KUKA KRL program: EPS_2_251806_MH01A_A_20260213065128.src

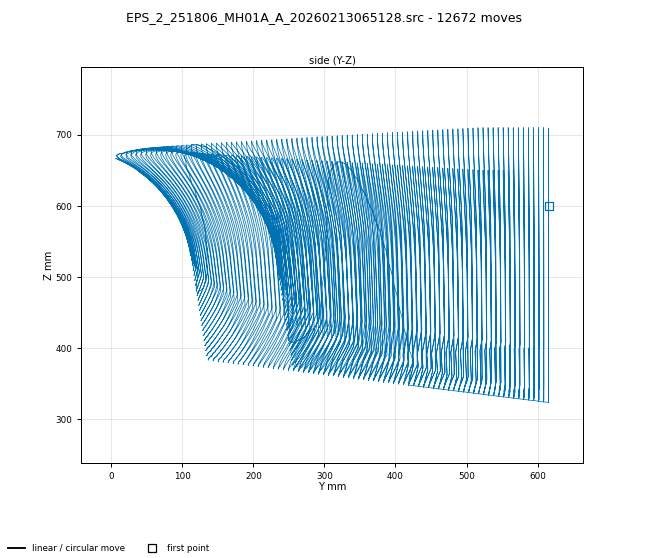
[picture p0: tool path of EPS_2_251806_MH01A_A_20260213065128.src, 12672 of 12674 moves have a stored position in this frame; points joined in program order, loops and branches not executed]
&ACCESS RVP
&REL 4
&COMMENT QRS 19112012
&PARAM EDITMASK = *
DEF PART()
EXT BAS (BAS_COMMAND :IN,REAL :IN )
INT I
BAS (#INITMOV,0 )

;KUKA QRS Post kuka4.cps  Date:22-06-2017 !

File_ID=3009

QRS_PRE_INIT()

;Init var - Until changes are made in qrs_pre_init
Outlet_Square_prg=0
Inlet_1_Square_prg=0
Inlet_2_Square_prg=0
Inlet_3_Square_prg=0
Inlet_4_Square_prg=0
Inlet_5_Square_prg=0

Outlet_1={X 0.000, Y 517.920, Z 561.000, B 0.000, E1 0.000 }
Inlet_1={X 0.000, Y 522.300, Z 501.000, B 0.000, E1 220.000 }
Outlet_1_type=299
Inlet_1_type=299
;QRS#1=Sidecore dimensions
;QRS#2=300-12" PVC SDR 35
;QRS#3=300-12" PVC SDR 35
;QRS#4=
;QRS#5=
;QRS#6=
;QRS#7=
;QRS#8=
;QRS#9=16M PSX
;QRS#10=16M PSX
;QRS#11=
;QRS#12=
;QRS#13=
;QRS#14=
;QRS#15=
;QRS#16=1220x127x991 3,25'
;QRS#17=EPS Height
;QRS#18=710,5
;QRS#19=*
;QRS#20= UPDATED VERSION 22-06-2017
;QRS#21=*
Outlet_Square=0150
Inlet_1_Square=0150
Inlet_2_Square=0
Inlet_3_Square=0
Inlet_4_Square=0
Inlet_5_Square=0
Mill_Square=1
Outlet_Square_Prg=206
Inlet_1_Square_prg=206

QRS_INIT()

$ADVANCE=5

; T1
PTP {E1 173.607,E2 173.607}
PTP {X 0,Y 615.503,A -85,B 0,C 180,E1 173.607,E2 173.607,E3 0,E4 0,E5 0,E6 0}
QRS_SPEED_INIT()
LIN {X 0,Y 615.503,Z 600,A -85,B 0,C 180,E1 173.607,E2 173.607,E3 0,E4 0,E5 0,E6 0} C_VEL
LIN {X 0,Y 615.503,Z 333.492,A -85,B 0,C 180,E1 173.607,E2 173.607} C_VEL
LIN {X 0,Y 615.503,Z 325.319,A -85,B 0,C 180,E1 173.607,E2 173.607} C_VEL
LIN {X 0,Y 615.485,Z 323.319,A -85,B 0,C 180,E1 173.421,E2 173.421} C_VEL
LIN {X 0,Y 615.473,Z 323.319,A -85,B 0,C 180,E1 170.801,E2 170.801} C_VEL
LIN {X 0,Y 615.487,Z 323.307,A -85,B 0,C 180,E1 168.139,E2 168.139} C_VEL
LIN {X 0,Y 615.487,Z 323.319,A -85,B 0,C 180,E1 165.451,E2 165.451} C_VEL
LIN {X 0,Y 615.467,Z 323.317,A -85,B 0,C 180,E1 162.729,E2 162.729} C_VEL
LIN {X 0,Y 615.489,Z 323.308,A -85,B 0,C 180,E1 159.967,E2 159.967} C_VEL
LIN {X 0,Y 615.489,Z 323.324,A -85,B 0,C 180,E1 157.155,E2 157.155} C_VEL
LIN {X 0,Y 615.466,Z 323.312,A -85,B 0,C 180,E1 154.435,E2 154.435} C_VEL
LIN {X 0,Y 615.489,Z 323.319,A -85,B 0,C 180,E1 151.549,E2 151.549} C_VEL
LIN {X 0,Y 615.465,Z 323.32,A -85,B 0,C 180,E1 148.917,E2 148.917} C_VEL
LIN {X 0,Y 615.462,Z 323.313,A -85,B 0,C 180,E1 146.469,E2 146.469} C_VEL
LIN {X 0,Y 615.482,Z 323.309,A -85,B 0,C 180,E1 144.166,E2 144.166} C_VEL
LIN {X 0,Y 615.488,Z 323.311,A -85,B 0,C 180,E1 141.931,E2 141.931} C_VEL
LIN {X 0,Y 615.487,Z 323.328,A -85,B 0,C 180,E1 139.393,E2 139.393} C_VEL
LIN {X 0,Y 615.455,Z 323.317,A -85,B 0,C 180,E1 136.752,E2 136.752} C_VEL
LIN {X 0,Y 615.487,Z 323.311,A -85,B 0,C 180,E1 133.997,E2 133.997} C_VEL
LIN {X 0,Y 615.464,Z 323.321,A -85,B 0,C 180,E1 131.091,E2 131.091} C_VEL
LIN {X 0,Y 615.454,Z 323.319,A -85,B 0,C 180,E1 128.906,E2 128.906} C_VEL
LIN {X 0,Y 615.459,Z 323.314,A -85,B 0,C 180,E1 126.426,E2 126.426} C_VEL
LIN {X 0,Y 615.498,Z 323.324,A -85,B 0,C 180,E1 123.535,E2 123.535} C_VEL
LIN {X 0,Y 615.449,Z 323.319,A -85,B 0,C 180,E1 120.921,E2 120.921} C_VEL
LIN {X 0,Y 615.455,Z 323.315,A -85,B 0,C 180,E1 118.444,E2 118.444} C_VEL
LIN {X 0,Y 615.499,Z 323.325,A -85,B 0,C 180,E1 115.57,E2 115.57} C_VEL
LIN {X 0,Y 615.443,Z 323.319,A -85,B 0,C 180,E1 112.846,E2 112.846} C_VEL
LIN {X 0,Y 615.447,Z 323.316,A -85,B 0,C 180,E1 110.546,E2 110.546} C_VEL
LIN {X 0,Y 615.494,Z 323.315,A -85,B 0,C 180,E1 107.956,E2 107.956} C_VEL
LIN {X 0,Y 615.455,Z 323.322,A -85,B 0,C 180,E1 105.227,E2 105.227} C_VEL
LIN {X 0,Y 615.451,Z 323.322,A -85,B 0,C 180,E1 103.202,E2 103.202} C_VEL
LIN {X 0,Y 615.434,Z 323.32,A -85,B 0,C 180,E1 100.86,E2 100.86} C_VEL
LIN {X 0,Y 615.444,Z 323.317,A -85,B 0,C 180,E1 98.537,E2 98.537} C_VEL
LIN {X 0,Y 615.497,Z 323.318,A -85,B 0,C 180,E1 95.898,E2 95.898} C_VEL
LIN {X 0,Y 615.448,Z 323.323,A -85,B 0,C 180,E1 93.273,E2 93.273} C_VEL
LIN {X 0,Y 615.449,Z 323.323,A -85,B 0,C 180,E1 91.308,E2 91.308} C_VEL
LIN {X 0,Y 615.451,Z 323.323,A -85,B 0,C 180,E1 89.345,E2 89.345} C_VEL
LIN {X 0,Y 615.452,Z 323.323,A -85,B 0,C 180,E1 87.382,E2 87.382} C_VEL
LIN {X 0,Y 615.454,Z 323.323,A -85,B 0,C 180,E1 85.415,E2 85.415} C_VEL
LIN {X 0,Y 615.455,Z 323.324,A -85,B 0,C 180,E1 83.443,E2 83.443} C_VEL
LIN {X 0,Y 615.455,Z 323.324,A -85,B 0,C 180,E1 81.463,E2 81.463} C_VEL
LIN {X 0,Y 615.429,Z 323.323,A -85,B 0,C 180,E1 79.143,E2 79.143} C_VEL
LIN {X 0,Y 615.424,Z 323.322,A -85,B 0,C 180,E1 76.797,E2 76.797} C_VEL
LIN {X 0,Y 615.479,Z 323.321,A -85,B 0,C 180,E1 74.094,E2 74.094} C_VEL
LIN {X 0,Y 615.435,Z 323.324,A -85,B 0,C 180,E1 71.352,E2 71.352} C_VEL
LIN {X 0,Y 615.433,Z 323.469,A -85,B 0,C 180,E1 70.552,E2 70.552} C_VEL
LIN {X 0,Y 615.467,Z 340.354,A -85,B 0,C 180,E1 68.193,E2 68.193} C_VEL
LIN {X 0,Y 615.47,Z 505.061,A -85,B 0,C 180,E1 66.189,E2 66.189} C_VEL
LIN {X 0,Y 615.489,Z 520.711,A -85,B 0,C 180,E1 65.86,E2 65.86} C_VEL
LIN {X 0,Y 615.479,Z 535.48,A -85,B 0,C 180,E1 65.413,E2 65.413} C_VEL
LIN {X 0,Y 615.487,Z 549.225,A -85,B 0,C 180,E1 64.865,E2 64.865} C_VEL
LIN {X 0,Y 615.482,Z 562.727,A -85,B 0,C 180,E1 64.193,E2 64.193} C_VEL
LIN {X 0,Y 615.496,Z 575.661,A -85,B 0,C 180,E1 63.406,E2 63.406} C_VEL
LIN {X 0,Y 615.494,Z 587.419,A -85,B 0,C 180,E1 62.547,E2 62.547} C_VEL
LIN {X 0,Y 615.496,Z 598.891,A -85,B 0,C 180,E1 61.549,E2 61.549} C_VEL
LIN {X 0,Y 615.495,Z 609.92,A -85,B 0,C 180,E1 60.399,E2 60.399} C_VEL
LIN {X 0,Y 615.497,Z 618.936,A -85,B 0,C 180,E1 59.271,E2 59.271} C_VEL
LIN {X 0,Y 615.493,Z 627.407,A -85,B 0,C 180,E1 57.992,E2 57.992} C_VEL
LIN {X 0,Y 615.493,Z 634.042,A -85,B 0,C 180,E1 56.764,E2 56.764} C_VEL
LIN {X 0,Y 615.496,Z 639.007,A -85,B 0,C 180,E1 55.64,E2 55.64} C_VEL
LIN {X 0,Y 615.496,Z 643.984,A -85,B 0,C 180,E1 54.166,E2 54.166} C_VEL
LIN {X 0,Y 615.491,Z 647.294,A -85,B 0,C 180,E1 52.758,E2 52.758} C_VEL
LIN {X 0,Y 615.495,Z 648.577,A -85,B 0,C 180,E1 51.932,E2 51.932} C_VEL
LIN {X 0,Y 615.49,Z 649.536,A -85,B 0,C 180,E1 50.938,E2 50.938} C_VEL
LIN {X 0,Y 615.498,Z 649.883,A -85,B 0,C 180,E1 49.91,E2 49.91} C_VEL
LIN {X 0,Y 615.491,Z 649.219,A -85,B 0,C 180,E1 48.526,E2 48.526} C_VEL
LIN {X 0,Y 615.49,Z 646.908,A -85,B 0,C 180,E1 46.953,E2 46.953} C_VEL
LIN {X 0,Y 615.493,Z 643.15,A -85,B 0,C 180,E1 45.461,E2 45.461} C_VEL
LIN {X 0,Y 615.496,Z 638.541,A -85,B 0,C 180,E1 44.149,E2 44.149} C_VEL
LIN {X 0,Y 615.49,Z 631.812,A -85,B 0,C 180,E1 42.7,E2 42.7} C_VEL
LIN {X 0,Y 615.494,Z 624.699,A -85,B 0,C 180,E1 41.474,E2 41.474} C_VEL
LIN {X 0,Y 615.496,Z 615.8,A -85,B 0,C 180,E1 40.219,E2 40.219} C_VEL
LIN {X 0,Y 615.495,Z 605.897,A -85,B 0,C 180,E1 39.063,E2 39.063} C_VEL
LIN {X 0,Y 615.496,Z 595.149,A -85,B 0,C 180,E1 38.013,E2 38.013} C_VEL
LIN {X 0,Y 615.495,Z 582.892,A -85,B 0,C 180,E1 37.013,E2 37.013} C_VEL
LIN {X 0,Y 615.497,Z 569.807,A -85,B 0,C 180,E1 36.129,E2 36.129} C_VEL
LIN {X 0,Y 615.476,Z 556.032,A -85,B 0,C 180,E1 35.366,E2 35.366} C_VEL
LIN {X 0,Y 615.492,Z 542.424,A -85,B 0,C 180,E1 34.758,E2 34.758} C_VEL
LIN {X 0,Y 615.486,Z 527.304,A -85,B 0,C 180,E1 34.234,E2 34.234} C_VEL
LIN {X 0,Y 615.48,Z 512.906,A -85,B 0,C 180,E1 33.868,E2 33.868} C_VEL
LIN {X 0,Y 615.461,Z 496.852,A -85,B 0,C 180,E1 33.605,E2 33.605} C_VEL
LIN {X 0,Y 615.465,Z 340.427,A -85,B 0,C 180,E1 31.727,E2 31.727} C_VEL
LIN {X 0,Y 615.421,Z 323.324,A -85,B 0,C 180,E1 29.328,E2 29.328} C_VEL
LIN {X 0,Y 615.415,Z 323.324,A -85,B 0,C 180,E1 27.031,E2 27.031} C_VEL
LIN {X 0,Y 615.475,Z 323.325,A -85,B 0,C 180,E1 24.273,E2 24.273} C_VEL
LIN {X 0,Y 615.433,Z 323.321,A -85,B 0,C 180,E1 21.434,E2 21.434} C_VEL
LIN {X 0,Y 615.43,Z 323.321,A -85,B 0,C 180,E1 19.34,E2 19.34} C_VEL
LIN {X 0,Y 615.429,Z 323.321,A -85,B 0,C 180,E1 17.272,E2 17.272} C_VEL
LIN {X 0,Y 615.43,Z 323.32,A -85,B 0,C 180,E1 15.228,E2 15.228} C_VEL
LIN {X 0,Y 615.432,Z 323.32,A -85,B 0,C 180,E1 13.203,E2 13.203} C_VEL
LIN {X 0,Y 615.47,Z 323.324,A -85,B 0,C 180,E1 10.527,E2 10.527} C_VEL
LIN {X 0,Y 615.48,Z 323.315,A -85,B 0,C 180,E1 7.876,E2 7.876} C_VEL
LIN {X 0,Y 615.439,Z 323.319,A -85,B 0,C 180,E1 5.242,E2 5.242} C_VEL
LIN {X 0,Y 615.475,Z 323.323,A -85,B 0,C 180,E1 2.618,E2 2.618} C_VEL
LIN {X 0,Y 615.486,Z 323.314,A -85,B 0,C 180,E1 0,E2 0} C_VEL
LIN {X 0,Y 615.45,Z 323.316,A -85,B 0,C 180,E1 -2.618,E2 -2.618} C_VEL
LIN {X 0,Y 615.474,Z 323.323,A -85,B 0,C 180,E1 -5.241,E2 -5.241} C_VEL
LIN {X 0,Y 615.493,Z 323.313,A -85,B 0,C 180,E1 -7.875,E2 -7.875} C_VEL
LIN {X 0,Y 615.458,Z 323.314,A -85,B 0,C 180,E1 -10.527,E2 -10.527} C_VEL
LIN {X 0,Y 615.483,Z 323.323,A -85,B 0,C 180,E1 -13.201,E2 -13.201} C_VEL
LIN {X 0,Y 615.491,Z 323.31,A -85,B 0,C 180,E1 -15.905,E2 -15.905} C_VEL
LIN {X 0,Y 615.462,Z 323.316,A -85,B 0,C 180,E1 -18.647,E2 -18.647} C_VEL
LIN {X 0,Y 615.489,Z 323.321,A -85,B 0,C 180,E1 -21.432,E2 -21.432} C_VEL
LIN {X 0,Y 615.477,Z 323.31,A -85,B 0,C 180,E1 -24.272,E2 -24.272} C_VEL
LIN {X 0,Y 615.487,Z 323.328,A -85,B 0,C 180,E1 -27.177,E2 -27.177} C_VEL
LIN {X 0,Y 615.486,Z 323.308,A -85,B 0,C 180,E1 -30.16,E2 -30.16} C_VEL
LIN {X 0,Y 615.474,Z 323.313,A -85,B 0,C 180,E1 -32.458,E2 -32.458} C_VEL
LIN {X 0,Y 615.477,Z 323.322,A -85,B 0,C 180,E1 -34.816,E2 -34.816} C_VEL
LIN {X 0,Y 615.485,Z 323.321,A -85,B 0,C 180,E1 -37.242,E2 -37.242} C_VEL
LIN {X 0,Y 615.493,Z 323.306,A -85,B 0,C 180,E1 -40.089,E2 -40.089} C_VEL
LIN {X 0,Y 615.49,Z 323.323,A -85,B 0,C 180,E1 -43.047,E2 -43.047} C_VEL
LIN {X 0,Y 615.487,Z 323.308,A -85,B 0,C 180,E1 -46.002,E2 -46.002} C_VEL
LIN {X 0,Y 615.485,Z 323.327,A -85,B 0,C 180,E1 -48.906,E2 -48.906} C_VEL
LIN {X 0,Y 615.478,Z 323.321,A -85,B 0,C 180,E1 -51.095,E2 -51.095} C_VEL
LIN {X 0,Y 615.469,Z 323.312,A -85,B 0,C 180,E1 -53.574,E2 -53.574} C_VEL
LIN {X 0,Y 615.488,Z 323.318,A -85,B 0,C 180,E1 -56.466,E2 -56.466} C_VEL
LIN {X 0,Y 615.469,Z 323.32,A -85,B 0,C 180,E1 -59.079,E2 -59.079} C_VEL
LIN {X 0,Y 615.464,Z 323.313,A -85,B 0,C 180,E1 -61.554,E2 -61.554} C_VEL
LIN {X 0,Y 615.478,Z 323.359,A -85,B 0,C 180,E1 -63.783,E2 -63.783} C_VEL
LIN {X 0,Y 615.479,Z 349.6,A -85,B 0,C 180,E1 -66.621,E2 -66.621} C_VEL
LIN {X 0,Y 615.488,Z 376.247,A -85,B 0,C 180,E1 -69.443,E2 -69.443} C_VEL
LIN {X 0,Y 615.496,Z 398.316,A -85,B 0,C 180,E1 -71.741,E2 -71.741} C_VEL
LIN {X 0,Y 615.481,Z 565.27,A -85,B 0,C 180,E1 -73.77,E2 -73.77} C_VEL
LIN {X 0,Y 615.49,Z 580.703,A -85,B 0,C 180,E1 -74.095,E2 -74.095} C_VEL
LIN {X 0,Y 615.48,Z 596.043,A -85,B 0,C 180,E1 -74.562,E2 -74.562} C_VEL
LIN {X 0,Y 615.484,Z 609.747,A -85,B 0,C 180,E1 -75.112,E2 -75.112} C_VEL
LIN {X 0,Y 615.493,Z 624.044,A -85,B 0,C 180,E1 -75.833,E2 -75.833} C_VEL
LIN {X 0,Y 615.497,Z 636.895,A -85,B 0,C 180,E1 -76.631,E2 -76.631} C_VEL
LIN {X 0,Y 615.495,Z 649.252,A -85,B 0,C 180,E1 -77.554,E2 -77.554} C_VEL
LIN {X 0,Y 615.495,Z 659.604,A -85,B 0,C 180,E1 -78.473,E2 -78.473} C_VEL
LIN {X 0,Y 615.494,Z 669.182,A -85,B 0,C 180,E1 -79.473,E2 -79.473} C_VEL
LIN {X 0,Y 615.493,Z 678.575,A -85,B 0,C 180,E1 -80.635,E2 -80.635} C_VEL
LIN {X 0,Y 615.497,Z 686.379,A -85,B 0,C 180,E1 -81.794,E2 -81.794} C_VEL
LIN {X 0,Y 615.494,Z 693.609,A -85,B 0,C 180,E1 -83.102,E2 -83.102} C_VEL
LIN {X 0,Y 615.499,Z 699.435,A -85,B 0,C 180,E1 -84.43,E2 -84.43} C_VEL
LIN {X 0,Y 615.491,Z 702.859,A -85,B 0,C 180,E1 -85.415,E2 -85.415} C_VEL
LIN {X 0,Y 615.493,Z 706.317,A -85,B 0,C 180,E1 -86.727,E2 -86.727} C_VEL
LIN {X 0,Y 615.499,Z 708.592,A -85,B 0,C 180,E1 -88.037,E2 -88.037} C_VEL
LIN {X 0,Y 615.491,Z 709.741,A -85,B 0,C 180,E1 -89.345,E2 -89.345} C_VEL
LIN {X 0,Y 615.491,Z 709.741,A -85,B 0,C 180,E1 -90.654,E2 -90.654} C_VEL
LIN {X 0,Y 615.499,Z 708.593,A -85,B 0,C 180,E1 -91.963,E2 -91.963} C_VEL
LIN {X 0,Y 615.493,Z 706.319,A -85,B 0,C 180,E1 -93.273,E2 -93.273} C_VEL
LIN {X 0,Y 615.491,Z 702.861,A -85,B 0,C 180,E1 -94.584,E2 -94.584} C_VEL
LIN {X 0,Y 615.497,Z 698.144,A -85,B 0,C 180,E1 -95.898,E2 -95.898} C_VEL
LIN {X 0,Y 615.492,Z 692.031,A -85,B 0,C 180,E1 -97.215,E2 -97.215} C_VEL
LIN {X 0,Y 615.49,Z 684.335,A -85,B 0,C 180,E1 -98.536,E2 -98.536} C_VEL
LIN {X 0,Y 615.495,Z 676.116,A -85,B 0,C 180,E1 -99.696,E2 -99.696} C_VEL
LIN {X 0,Y 615.496,Z 665.898,A -85,B 0,C 180,E1 -100.892,E2 -100.892} C_VEL
LIN {X 0,Y 615.496,Z 656.07,A -85,B 0,C 180,E1 -101.86,E2 -101.86} C_VEL
LIN {X 0,Y 615.497,Z 643.951,A -85,B 0,C 180,E1 -102.865,E2 -102.865} C_VEL
LIN {X 0,Y 615.498,Z 631.802,A -85,B 0,C 180,E1 -103.705,E2 -103.705} C_VEL
LIN {X 0,Y 615.477,Z 618.384,A -85,B 0,C 180,E1 -104.472,E2 -104.472} C_VEL
LIN {X 0,Y 615.495,Z 603.855,A -85,B 0,C 180,E1 -105.141,E2 -105.141} C_VEL
LIN {X 0,Y 615.48,Z 589.625,A -85,B 0,C 180,E1 -105.65,E2 -105.65} C_VEL
LIN {X 0,Y 615.5,Z 575.177,A -85,B 0,C 180,E1 -106.035,E2 -106.035} C_VEL
LIN {X 0,Y 615.478,Z 560.741,A -85,B 0,C 180,E1 -106.296,E2 -106.296} C_VEL
LIN {X 0,Y 615.495,Z 398.319,A -85,B 0,C 180,E1 -108.259,E2 -108.259} C_VEL
LIN {X 0,Y 615.484,Z 372.931,A -85,B 0,C 180,E1 -110.905,E2 -110.905} C_VEL
LIN {X 0,Y 615.477,Z 346.881,A -85,B 0,C 180,E1 -113.67,E2 -113.67} C_VEL
LIN {X 0,Y 615.477,Z 323.365,A -85,B 0,C 180,E1 -116.216,E2 -116.216} C_VEL
LIN {X 0,Y 615.458,Z 323.316,A -85,B 0,C 180,E1 -118.659,E2 -118.659} C_VEL
LIN {X 0,Y 615.476,Z 323.322,A -85,B 0,C 180,E1 -121.084,E2 -121.084} C_VEL
LIN {X 0,Y 615.492,Z 323.308,A -85,B 0,C 180,E1 -124.021,E2 -124.021} C_VEL
LIN {X 0,Y 615.466,Z 323.312,A -85,B 0,C 180,E1 -126.426,E2 -126.426} C_VEL
LIN {X 0,Y 615.48,Z 323.322,A -85,B 0,C 180,E1 -129.061,E2 -129.061} C_VEL
LIN {X 0,Y 615.489,Z 323.319,A -85,B 0,C 180,E1 -131.473,E2 -131.473} C_VEL
LIN {X 0,Y 615.485,Z 323.308,A -85,B 0,C 180,E1 -134.149,E2 -134.149} C_VEL
LIN {X 0,Y 615.477,Z 323.321,A -85,B 0,C 180,E1 -136.953,E2 -136.953} C_VEL
LIN {X 0,Y 615.494,Z 323.307,A -85,B 0,C 180,E1 -139.91,E2 -139.91} C_VEL
LIN {X 0,Y 615.471,Z 323.318,A -85,B 0,C 180,E1 -142.757,E2 -142.757} C_VEL
LIN {X 0,Y 615.491,Z 323.322,A -85,B 0,C 180,E1 -145.298,E2 -145.298} C_VEL
LIN {X 0,Y 615.481,Z 323.313,A -85,B 0,C 180,E1 -147.669,E2 -147.669} C_VEL
LIN {X 0,Y 615.483,Z 323.308,A -85,B 0,C 180,E1 -150.205,E2 -150.205} C_VEL
LIN {X 0,Y 615.488,Z 323.322,A -85,B 0,C 180,E1 -152.954,E2 -152.954} C_VEL
LIN {X 0,Y 615.484,Z 323.31,A -85,B 0,C 180,E1 -155.728,E2 -155.728} C_VEL
LIN {X 0,Y 615.474,Z 323.316,A -85,B 0,C 180,E1 -158.568,E2 -158.568} C_VEL
LIN {X 0,Y 615.48,Z 323.317,A -85,B 0,C 180,E1 -161.396,E2 -161.396} C_VEL
LIN {X 0,Y 615.487,Z 323.307,A -85,B 0,C 180,E1 -164.095,E2 -164.095} C_VEL
LIN {X 0,Y 615.484,Z 323.321,A -85,B 0,C 180,E1 -166.799,E2 -166.799} C_VEL
LIN {X 0,Y 615.476,Z 323.315,A -85,B 0,C 180,E1 -169.473,E2 -169.473} C_VEL
LIN {X 0,Y 615.488,Z 323.307,A -85,B 0,C 180,E1 -172.125,E2 -172.125} C_VEL
LIN {X 0,Y 615.485,Z 323.322,A -85,B 0,C 180,E1 -174.759,E2 -174.759} C_VEL
LIN {X 0,Y 615.474,Z 323.316,A -85,B 0,C 180,E1 -177.382,E2 -177.382} C_VEL
LIN {X 0,Y 615.486,Z 323.308,A -85,B 0,C 180,E1 -180,E2 -180} C_VEL
LIN {X 0,Y 615.483,Z 323.319,A -85,B 0,C 180,E1 -182.618,E2 -182.618} C_VEL
LIN {X 0,Y 615.474,Z 323.318,A -85,B 0,C 180,E1 -185.242,E2 -185.242} C_VEL
LIN {X 0,Y 615.485,Z 323.319,A -85,B 0,C 180,E1 -186.579,E2 -186.579} C_VEL
LIN {X 0,Y 614.801,Z 323.467,A -85,B 0,C 180,E1 -187.125,E2 -187.125} C_VEL
LIN {X 0,Y 611.96,Z 323.875,A -85,B 0,C 180,E1 -188.011,E2 -188.011} C_VEL
LIN {X 0,Y 609.569,Z 324.187,A -85,B 0,C 180,E1 -188.724,E2 -188.724} C_VEL
LIN {X 0,Y 608.539,Z 324.305,A -85,B 0,C 180,E1 -189.274,E2 -189.274} C_VEL
LIN {X 0,Y 608.452,Z 324.314,A -85,B 0,C 180,E1 -189.46,E2 -189.46} C_VEL
LIN {X 0,Y 608.462,Z 324.311,A -85,B 0,C 180,E1 -192,E2 -192} C_VEL
LIN {X 0,Y 608.471,Z 324.319,A -85,B 0,C 180,E1 -194.721,E2 -194.721} C_VEL
LIN {X 0,Y 608.442,Z 324.314,A -85,B 0,C 180,E1 -197.477,E2 -197.477} C_VEL
LIN {X 0,Y 608.463,Z 324.314,A -85,B 0,C 180,E1 -200.274,E2 -200.274} C_VEL
LIN {X 0,Y 608.445,Z 324.317,A -85,B 0,C 180,E1 -203.125,E2 -203.125} C_VEL
LIN {X 0,Y 608.457,Z 324.312,A -85,B 0,C 180,E1 -205.719,E2 -205.719} C_VEL
LIN {X 0,Y 608.475,Z 324.319,A -85,B 0,C 180,E1 -208.621,E2 -208.621} C_VEL
LIN {X 0,Y 608.439,Z 324.315,A -85,B 0,C 180,E1 -211.319,E2 -211.319} C_VEL
LIN {X 0,Y 608.445,Z 324.313,A -85,B 0,C 180,E1 -213.732,E2 -213.732} C_VEL
LIN {X 0,Y 608.477,Z 324.311,A -85,B 0,C 180,E1 -216.091,E2 -216.091} C_VEL
LIN {X 0,Y 608.462,Z 324.321,A -85,B 0,C 180,E1 -218.589,E2 -218.589} C_VEL
LIN {X 0,Y 608.437,Z 324.315,A -85,B 0,C 180,E1 -221.34,E2 -221.34} C_VEL
LIN {X 0,Y 608.46,Z 324.316,A -85,B 0,C 180,E1 -224.265,E2 -224.265} C_VEL
LIN {X 0,Y 608.43,Z 324.318,A -85,B 0,C 180,E1 -227.039,E2 -227.039} C_VEL
LIN {X 0,Y 608.454,Z 324.312,A -85,B 0,C 180,E1 -229.697,E2 -229.697} C_VEL
LIN {X 0,Y 608.464,Z 324.317,A -85,B 0,C 180,E1 -232.254,E2 -232.254} C_VEL
LIN {X 0,Y 608.42,Z 324.318,A -85,B 0,C 180,E1 -235.099,E2 -235.099} C_VEL
LIN {X 0,Y 608.436,Z 324.314,A -85,B 0,C 180,E1 -237.482,E2 -237.482} C_VEL
LIN {X 0,Y 608.479,Z 324.315,A -85,B 0,C 180,E1 -240.221,E2 -240.221} C_VEL
LIN {X 0,Y 608.416,Z 324.317,A -85,B 0,C 180,E1 -243.225,E2 -243.225} C_VEL
LIN {X 0,Y 608.431,Z 324.315,A -85,B 0,C 180,E1 -245.428,E2 -245.428} C_VEL
LIN {X 0,Y 608.464,Z 324.32,A -85,B 0,C 180,E1 -248.309,E2 -248.309} C_VEL
LIN {X 0,Y 608.436,Z 324.315,A -85,B 0,C 180,E1 -251.13,E2 -251.13} C_VEL
LIN {X 0,Y 608.454,Z 324.315,A -85,B 0,C 180,E1 -253.906,E2 -253.906} C_VEL
LIN {X 0,Y 608.44,Z 324.319,A -85,B 0,C 180,E1 -256.643,E2 -256.643} C_VEL
LIN {X 0,Y 608.406,Z 324.319,A -85,B 0,C 180,E1 -259.078,E2 -259.078} C_VEL
LIN {X 0,Y 608.419,Z 324.316,A -85,B 0,C 180,E1 -261.364,E2 -261.364} C_VEL
LIN {X 0,Y 608.464,Z 324.317,A -85,B 0,C 180,E1 -264.033,E2 -264.033} C_VEL
LIN {X 0,Y 608.42,Z 324.32,A -85,B 0,C 180,E1 -266.689,E2 -266.689} C_VEL
LIN {X 0,Y 608.438,Z 324.318,A -85,B 0,C 180,E1 -268.677,E2 -268.677} C_VEL
LIN {X 0,Y 608.449,Z 324.317,A -85,B 0,C 180,E1 -270.662,E2 -270.662} C_VEL
LIN {X 0,Y 608.403,Z 324.318,A -85,B 0,C 180,E1 -273.311,E2 -273.311} C_VEL
LIN {X 0,Y 608.455,Z 324.318,A -85,B 0,C 180,E1 -275.967,E2 -275.967} C_VEL
LIN {X 0,Y 608.425,Z 324.319,A -85,B 0,C 180,E1 -278.637,E2 -278.637} C_VEL
LIN {X 0,Y 608.413,Z 324.317,A -85,B 0,C 180,E1 -281.325,E2 -281.325} C_VEL
LIN {X 0,Y 608.474,Z 324.318,A -85,B 0,C 180,E1 -284.038,E2 -284.038} C_VEL
LIN {X 0,Y 608.412,Z 324.319,A -85,B 0,C 180,E1 -286.785,E2 -286.785} C_VEL
LIN {X 0,Y 608.431,Z 324.391,A -85,B 0,C 180,E1 -289.33,E2 -289.33} C_VEL
LIN {X 0,Y 608.497,Z 340.471,A -85,B 0,C 180,E1 -291.602,E2 -291.602} C_VEL
LIN {X 0,Y 608.726,Z 347.856,A -85,B 0,C 180,E1 -291.704,E2 -291.704} C_VEL
LIN {X 0,Y 608.67,Z 504.169,A -85,B 0,C 180,E1 -293.611,E2 -293.611} C_VEL
LIN {X 0,Y 608.67,Z 519.292,A -85,B 0,C 180,E1 -293.922,E2 -293.922} C_VEL
LIN {X 0,Y 608.621,Z 534.552,A -85,B 0,C 180,E1 -294.377,E2 -294.377} C_VEL
LIN {X 0,Y 608.595,Z 548.477,A -85,B 0,C 180,E1 -294.93,E2 -294.93} C_VEL
LIN {X 0,Y 608.549,Z 562.697,A -85,B 0,C 180,E1 -295.639,E2 -295.639} C_VEL
LIN {X 0,Y 608.539,Z 575.141,A -85,B 0,C 180,E1 -296.4,E2 -296.4} C_VEL
LIN {X 0,Y 608.529,Z 587.705,A -85,B 0,C 180,E1 -297.323,E2 -297.323} C_VEL
LIN {X 0,Y 608.485,Z 598.502,A -85,B 0,C 180,E1 -298.265,E2 -298.265} C_VEL
LIN {X 0,Y 608.484,Z 609.414,A -85,B 0,C 180,E1 -299.398,E2 -299.398} C_VEL
LIN {X 0,Y 608.453,Z 618.668,A -85,B 0,C 180,E1 -300.546,E2 -300.546} C_VEL
LIN {X 0,Y 608.462,Z 626.497,A -85,B 0,C 180,E1 -301.705,E2 -301.705} C_VEL
LIN {X 0,Y 608.443,Z 633.127,A -85,B 0,C 180,E1 -302.881,E2 -302.881} C_VEL
LIN {X 0,Y 608.44,Z 638.579,A -85,B 0,C 180,E1 -304.071,E2 -304.071} C_VEL
LIN {X 0,Y 608.424,Z 642.975,A -85,B 0,C 180,E1 -305.279,E2 -305.279} C_VEL
LIN {X 0,Y 608.424,Z 645.349,A -85,B 0,C 180,E1 -306.094,E2 -306.094} C_VEL
LIN {X 0,Y 608.432,Z 647.777,A -85,B 0,C 180,E1 -307.153,E2 -307.153} C_VEL
LIN {X 0,Y 608.413,Z 649.814,A -85,B 0,C 180,E1 -308.592,E2 -308.592} C_VEL
LIN {X 0,Y 608.412,Z 650.365,A -85,B 0,C 180,E1 -309.444,E2 -309.444} C_VEL
LIN {X 0,Y 608.437,Z 650.44,A -85,B 0,C 180,E1 -310.327,E2 -310.327} C_VEL
LIN {X 0,Y 608.415,Z 649.935,A -85,B 0,C 180,E1 -311.337,E2 -311.337} C_VEL
LIN {X 0,Y 608.434,Z 648.787,A -85,B 0,C 180,E1 -312.331,E2 -312.331} C_VEL
LIN {X 0,Y 608.433,Z 646.997,A -85,B 0,C 180,E1 -313.305,E2 -313.305} C_VEL
LIN {X 0,Y 608.423,Z 643.011,A -85,B 0,C 180,E1 -314.799,E2 -314.799} C_VEL
LIN {X 0,Y 608.431,Z 638.119,A -85,B 0,C 180,E1 -316.127,E2 -316.127} C_VEL
LIN {X 0,Y 608.438,Z 632.233,A -85,B 0,C 180,E1 -317.38,E2 -317.38} C_VEL
LIN {X 0,Y 608.443,Z 624.795,A -85,B 0,C 180,E1 -318.66,E2 -318.66} C_VEL
LIN {X 0,Y 608.474,Z 615.89,A -85,B 0,C 180,E1 -319.915,E2 -319.915} C_VEL
LIN {X 0,Y 608.494,Z 606.133,A -85,B 0,C 180,E1 -321.058,E2 -321.058} C_VEL
LIN {X 0,Y 608.497,Z 595.21,A -85,B 0,C 180,E1 -322.132,E2 -322.132} C_VEL
LIN {X 0,Y 608.519,Z 583.62,A -85,B 0,C 180,E1 -323.089,E2 -323.089} C_VEL
LIN {X 0,Y 608.548,Z 571.328,A -85,B 0,C 180,E1 -323.942,E2 -323.942} C_VEL
LIN {X 0,Y 608.576,Z 557.514,A -85,B 0,C 180,E1 -324.731,E2 -324.731} C_VEL
LIN {X 0,Y 608.622,Z 543.682,A -85,B 0,C 180,E1 -325.368,E2 -325.368} C_VEL
LIN {X 0,Y 608.637,Z 529.142,A -85,B 0,C 180,E1 -325.892,E2 -325.892} C_VEL
LIN {X 0,Y 608.654,Z 513.527,A -85,B 0,C 180,E1 -326.304,E2 -326.304} C_VEL
LIN {X 0,Y 608.658,Z 497.334,A -85,B 0,C 180,E1 -326.577,E2 -326.577} C_VEL
LIN {X 0,Y 608.598,Z 341.195,A -85,B 0,C 180,E1 -328.471,E2 -328.471} C_VEL
LIN {X 0,Y 608.47,Z 340.371,A -85,B 0,C 180,E1 -328.503,E2 -328.503} C_VEL
LIN {X 0,Y 608.414,Z 324.367,A -85,B 0,C 180,E1 -330.764,E2 -330.764} C_VEL
LIN {X 0,Y 608.391,Z 324.321,A -85,B 0,C 180,E1 -333.223,E2 -333.223} C_VEL
LIN {X 0,Y 608.456,Z 324.323,A -85,B 0,C 180,E1 -335.853,E2 -335.853} C_VEL
LIN {X 0,Y 608.441,Z 324.317,A -85,B 0,C 180,E1 -338.307,E2 -338.307} C_VEL
LIN {X 0,Y 608.428,Z 324.316,A -85,B 0,C 180,E1 -341.129,E2 -341.129} C_VEL
LIN {X 0,Y 608.454,Z 324.321,A -85,B 0,C 180,E1 -343.906,E2 -343.906} C_VEL
LIN {X 0,Y 608.424,Z 324.316,A -85,B 0,C 180,E1 -346.642,E2 -346.642} C_VEL
LIN {X 0,Y 608.439,Z 324.319,A -85,B 0,C 180,E1 -349.349,E2 -349.349} C_VEL
LIN {X 0,Y 608.472,Z 324.314,A -85,B 0,C 180,E1 -352.033,E2 -352.033} C_VEL
LIN {X 0,Y 608.425,Z 324.316,A -85,B 0,C 180,E1 -354.698,E2 -354.698} C_VEL
LIN {X 0,Y 608.465,Z 324.317,A -85,B 0,C 180,E1 -357.352,E2 -357.352} C_VEL
LIN {X 0,Y 608.477,Z 324.313,A -85,B 0,C 180,E1 -360,E2 -360} C_VEL
LIN {X 0,Y 608.445,Z 324.313,A -85,B 0,C 180,E1 -362.648,E2 -362.648} C_VEL
LIN {X 0,Y 608.456,Z 324.32,A -85,B 0,C 180,E1 -365.302,E2 -365.302} C_VEL
LIN {X 0,Y 608.48,Z 324.311,A -85,B 0,C 180,E1 -367.967,E2 -367.967} C_VEL
LIN {X 0,Y 608.438,Z 324.315,A -85,B 0,C 180,E1 -370.65,E2 -370.65} C_VEL
LIN {X 0,Y 608.463,Z 324.322,A -85,B 0,C 180,E1 -373.356,E2 -373.356} C_VEL
LIN {X 0,Y 608.456,Z 324.312,A -85,B 0,C 180,E1 -376.094,E2 -376.094} C_VEL
LIN {X 0,Y 608.448,Z 324.317,A -85,B 0,C 180,E1 -378.87,E2 -378.87} C_VEL
LIN {X 0,Y 608.471,Z 324.313,A -85,B 0,C 180,E1 -381.691,E2 -381.691} C_VEL
LIN {X 0,Y 608.448,Z 324.314,A -85,B 0,C 180,E1 -384.571,E2 -384.571} C_VEL
LIN {X 0,Y 608.481,Z 324.319,A -85,B 0,C 180,E1 -387.207,E2 -387.207} C_VEL
LIN {X 0,Y 608.468,Z 324.311,A -85,B 0,C 180,E1 -389.971,E2 -389.971} C_VEL
LIN {X 0,Y 608.452,Z 324.319,A -85,B 0,C 180,E1 -392.88,E2 -392.88} C_VEL
LIN {X 0,Y 608.437,Z 324.321,A -85,B 0,C 180,E1 -395.278,E2 -395.278} C_VEL
LIN {X 0,Y 608.469,Z 324.311,A -85,B 0,C 180,E1 -397.746,E2 -397.746} C_VEL
LIN {X 0,Y 608.451,Z 324.314,A -85,B 0,C 180,E1 -400.329,E2 -400.329} C_VEL
LIN {X 0,Y 608.456,Z 324.323,A -85,B 0,C 180,E1 -402.959,E2 -402.959} C_VEL
LIN {X 0,Y 608.457,Z 324.312,A -85,B 0,C 180,E1 -405.736,E2 -405.736} C_VEL
LIN {X 0,Y 608.46,Z 324.319,A -85,B 0,C 180,E1 -408.658,E2 -408.658} C_VEL
LIN {X 0,Y 608.436,Z 324.316,A -85,B 0,C 180,E1 -411.409,E2 -411.409} C_VEL
LIN {X 0,Y 608.448,Z 324.313,A -85,B 0,C 180,E1 -413.954,E2 -413.954} C_VEL
LIN {X 0,Y 608.466,Z 324.314,A -85,B 0,C 180,E1 -416.329,E2 -416.329} C_VEL
LIN {X 0,Y 608.447,Z 324.324,A -85,B 0,C 180,E1 -418.732,E2 -418.732} C_VEL
LIN {X 0,Y 608.453,Z 324.314,A -85,B 0,C 180,E1 -421.383,E2 -421.383} C_VEL
LIN {X 0,Y 608.449,Z 324.401,A -85,B 0,C 180,E1 -423.572,E2 -423.572} C_VEL
LIN {X 0,Y 608.734,Z 329.1,A -85,B 0,C 180,E1 -424.105,E2 -424.105} C_VEL
LIN {X 0,Y 608.661,Z 354.598,A -85,B 0,C 180,E1 -426.884,E2 -426.884} C_VEL
LIN {X 0,Y 608.609,Z 381.255,A -85,B 0,C 180,E1 -429.731,E2 -429.731} C_VEL
LIN {X 0,Y 608.583,Z 398.319,A -85,B 0,C 180,E1 -431.526,E2 -431.526} C_VEL
LIN {X 0,Y 608.761,Z 403.953,A -85,B 0,C 180,E1 -431.613,E2 -431.613} C_VEL
LIN {X 0,Y 608.675,Z 565.269,A -85,B 0,C 180,E1 -433.583,E2 -433.583} C_VEL
LIN {X 0,Y 608.651,Z 580.702,A -85,B 0,C 180,E1 -433.911,E2 -433.911} C_VEL
LIN {X 0,Y 608.618,Z 596.042,A -85,B 0,C 180,E1 -434.383,E2 -434.383} C_VEL
LIN {X 0,Y 608.605,Z 609.75,A -85,B 0,C 180,E1 -434.94,E2 -434.94} C_VEL
LIN {X 0,Y 608.572,Z 623.231,A -85,B 0,C 180,E1 -435.624,E2 -435.624} C_VEL
LIN {X 0,Y 608.554,Z 635.66,A -85,B 0,C 180,E1 -436.39,E2 -436.39} C_VEL
LIN {X 0,Y 608.528,Z 648.28,A -85,B 0,C 180,E1 -437.324,E2 -437.324} C_VEL
LIN {X 0,Y 608.496,Z 659.745,A -85,B 0,C 180,E1 -438.339,E2 -438.339} C_VEL
LIN {X 0,Y 608.475,Z 669.386,A -85,B 0,C 180,E1 -439.35,E2 -439.35} C_VEL
LIN {X 0,Y 608.476,Z 678.852,A -85,B 0,C 180,E1 -440.526,E2 -440.526} C_VEL
LIN {X 0,Y 608.457,Z 686.728,A -85,B 0,C 180,E1 -441.698,E2 -441.698} C_VEL
LIN {X 0,Y 608.44,Z 694.086,A -85,B 0,C 180,E1 -443.034,E2 -443.034} C_VEL
LIN {X 0,Y 608.45,Z 699.923,A -85,B 0,C 180,E1 -444.365,E2 -444.365} C_VEL
LIN {X 0,Y 608.427,Z 703.382,A -85,B 0,C 180,E1 -445.362,E2 -445.362} C_VEL
LIN {X 0,Y 608.421,Z 706.885,A -85,B 0,C 180,E1 -446.689,E2 -446.689} C_VEL
LIN {X 0,Y 608.444,Z 709.191,A -85,B 0,C 180,E1 -448.014,E2 -448.014} C_VEL
LIN {X 0,Y 608.434,Z 710.35,A -85,B 0,C 180,E1 -449.338,E2 -449.338} C_VEL
LIN {X 0,Y 608.434,Z 710.351,A -85,B 0,C 180,E1 -450.662,E2 -450.662} C_VEL
LIN {X 0,Y 608.444,Z 709.192,A -85,B 0,C 180,E1 -451.986,E2 -451.986} C_VEL
LIN {X 0,Y 608.421,Z 706.886,A -85,B 0,C 180,E1 -453.311,E2 -453.311} C_VEL
LIN {X 0,Y 608.427,Z 703.384,A -85,B 0,C 180,E1 -454.638,E2 -454.638} C_VEL
LIN {X 0,Y 608.435,Z 698.609,A -85,B 0,C 180,E1 -455.967,E2 -455.967} C_VEL
LIN {X 0,Y 608.456,Z 692.427,A -85,B 0,C 180,E1 -457.299,E2 -457.299} C_VEL
LIN {X 0,Y 608.464,Z 684.656,A -85,B 0,C 180,E1 -458.636,E2 -458.636} C_VEL
LIN {X 0,Y 608.471,Z 676.373,A -85,B 0,C 180,E1 -459.809,E2 -459.809} C_VEL
LIN {X 0,Y 608.492,Z 665.653,A -85,B 0,C 180,E1 -461.063,E2 -461.063} C_VEL
LIN {X 0,Y 608.523,Z 654.278,A -85,B 0,C 180,E1 -462.167,E2 -462.167} C_VEL
LIN {X 0,Y 608.547,Z 642.858,A -85,B 0,C 180,E1 -463.099,E2 -463.099} C_VEL
LIN {X 0,Y 608.562,Z 630.452,A -85,B 0,C 180,E1 -463.95,E2 -463.95} C_VEL
LIN {X 0,Y 608.56,Z 616.865,A -85,B 0,C 180,E1 -464.718,E2 -464.718} C_VEL
LIN {X 0,Y 608.631,Z 602.799,A -85,B 0,C 180,E1 -465.359,E2 -465.359} C_VEL
LIN {X 0,Y 608.634,Z 588.311,A -85,B 0,C 180,E1 -465.874,E2 -465.874} C_VEL
LIN {X 0,Y 608.68,Z 573.07,A -85,B 0,C 180,E1 -466.269,E2 -466.269} C_VEL
LIN {X 0,Y 608.68,Z 557.237,A -85,B 0,C 180,E1 -466.532,E2 -466.532} C_VEL
LIN {X 0,Y 608.65,Z 398.951,A -85,B 0,C 180,E1 -468.451,E2 -468.451} C_VEL
LIN {X 0,Y 608.571,Z 398.127,A -85,B 0,C 180,E1 -468.495,E2 -468.495} C_VEL
LIN {X 0,Y 608.62,Z 372.931,A -85,B 0,C 180,E1 -471.152,E2 -471.152} C_VEL
LIN {X 0,Y 608.699,Z 345.819,A -85,B 0,C 180,E1 -474.065,E2 -474.065} C_VEL
LIN {X 0,Y 608.748,Z 326.281,A -85,B 0,C 180,E1 -476.205,E2 -476.205} C_VEL
LIN {X 0,Y 608.442,Z 324.316,A -85,B 0,C 180,E1 -476.45,E2 -476.45} C_VEL
LIN {X 0,Y 608.432,Z 324.32,A -85,B 0,C 180,E1 -479.021,E2 -479.021} C_VEL
LIN {X 0,Y 608.458,Z 324.323,A -85,B 0,C 180,E1 -481.317,E2 -481.317} C_VEL
LIN {X 0,Y 608.477,Z 324.313,A -85,B 0,C 180,E1 -483.736,E2 -483.736} C_VEL
LIN {X 0,Y 608.457,Z 324.312,A -85,B 0,C 180,E1 -486.091,E2 -486.091} C_VEL
LIN {X 0,Y 608.459,Z 324.313,A -85,B 0,C 180,E1 -488.588,E2 -488.588} C_VEL
LIN {X 0,Y 608.461,Z 324.32,A -85,B 0,C 180,E1 -491.342,E2 -491.342} C_VEL
LIN {X 0,Y 608.471,Z 324.311,A -85,B 0,C 180,E1 -493.869,E2 -493.869} C_VEL
LIN {X 0,Y 608.458,Z 324.314,A -85,B 0,C 180,E1 -496.692,E2 -496.692} C_VEL
LIN {X 0,Y 608.443,Z 324.318,A -85,B 0,C 180,E1 -498.823,E2 -498.823} C_VEL
LIN {X 0,Y 608.466,Z 324.312,A -85,B 0,C 180,E1 -501.759,E2 -501.759} C_VEL
LIN {X 0,Y 608.439,Z 324.317,A -85,B 0,C 180,E1 -504.722,E2 -504.722} C_VEL
LIN {X 0,Y 608.458,Z 324.316,A -85,B 0,C 180,E1 -507.478,E2 -507.478} C_VEL
LIN {X 0,Y 608.467,Z 324.31,A -85,B 0,C 180,E1 -510.221,E2 -510.221} C_VEL
LIN {X 0,Y 608.475,Z 324.315,A -85,B 0,C 180,E1 -512.793,E2 -512.793} C_VEL
LIN {X 0,Y 608.453,Z 324.317,A -85,B 0,C 180,E1 -515.429,E2 -515.429} C_VEL
LIN {X 0,Y 608.463,Z 324.311,A -85,B 0,C 180,E1 -518.308,E2 -518.308} C_VEL
LIN {X 0,Y 608.467,Z 324.317,A -85,B 0,C 180,E1 -521.284,E2 -521.284} C_VEL
LIN {X 0,Y 608.458,Z 324.312,A -85,B 0,C 180,E1 -523.906,E2 -523.906} C_VEL
LIN {X 0,Y 608.463,Z 324.316,A -85,B 0,C 180,E1 -526.644,E2 -526.644} C_VEL
LIN {X 0,Y 608.458,Z 324.316,A -85,B 0,C 180,E1 -529.35,E2 -529.35} C_VEL
LIN {X 0,Y 608.478,Z 324.309,A -85,B 0,C 180,E1 -532.033,E2 -532.033} C_VEL
LIN {X 0,Y 608.465,Z 324.317,A -85,B 0,C 180,E1 -534.698,E2 -534.698} C_VEL
LIN {X 0,Y 608.466,Z 324.314,A -85,B 0,C 180,E1 -537.352,E2 -537.352} C_VEL
LIN {X 0,Y 608.477,Z 324.309,A -85,B 0,C 180,E1 -540,E2 -540} C_VEL
LIN {X 0,Y 608.473,Z 324.316,A -85,B 0,C 180,E1 -542.648,E2 -542.648} C_VEL
LIN {X 0,Y 608.455,Z 324.315,A -85,B 0,C 180,E1 -545.302,E2 -545.302} C_VEL
LIN {X 0,Y 608.477,Z 324.309,A -85,B 0,C 180,E1 -547.967,E2 -547.967} C_VEL
LIN {X 0,Y 608.452,Z 324.314,A -85,B 0,C 180,E1 -549.46,E2 -549.46} C_VEL
LIN {X 0,Y 607.778,Z 324.398,A -85,B 0,C 180,E1 -550.012,E2 -550.012} C_VEL
LIN {X 0,Y 604.928,Z 324.761,A -85,B 0,C 180,E1 -550.909,E2 -550.909} C_VEL
LIN {X 0,Y 602.525,Z 325.055,A -85,B 0,C 180,E1 -551.631,E2 -551.631} C_VEL
LIN {X 0,Y 601.492,Z 325.181,A -85,B 0,C 180,E1 -552.187,E2 -552.187} C_VEL
LIN {X 0,Y 601.408,Z 325.193,A -85,B 0,C 180,E1 -552.376,E2 -552.376} C_VEL
LIN {X 0,Y 601.425,Z 325.197,A -85,B 0,C 180,E1 -554.897,E2 -554.897} C_VEL
LIN {X 0,Y 601.428,Z 325.194,A -85,B 0,C 180,E1 -556.986,E2 -556.986} C_VEL
LIN {X 0,Y 601.4,Z 325.191,A -85,B 0,C 180,E1 -559.81,E2 -559.81} C_VEL
LIN {X 0,Y 601.414,Z 325.197,A -85,B 0,C 180,E1 -562.606,E2 -562.606} C_VEL
LIN {X 0,Y 601.394,Z 325.199,A -85,B 0,C 180,E1 -564.879,E2 -564.879} C_VEL
LIN {X 0,Y 601.394,Z 325.193,A -85,B 0,C 180,E1 -567.359,E2 -567.359} C_VEL
LIN {X 0,Y 601.413,Z 325.19,A -85,B 0,C 180,E1 -569.394,E2 -569.394} C_VEL
LIN {X 0,Y 601.398,Z 325.191,A -85,B 0,C 180,E1 -571.728,E2 -571.728} C_VEL
LIN {X 0,Y 601.421,Z 325.19,A -85,B 0,C 180,E1 -574.119,E2 -574.119} C_VEL
LIN {X 0,Y 601.406,Z 325.2,A -85,B 0,C 180,E1 -576.583,E2 -576.583} C_VEL
LIN {X 0,Y 601.399,Z 325.194,A -85,B 0,C 180,E1 -579.128,E2 -579.128} C_VEL
LIN {X 0,Y 601.421,Z 325.188,A -85,B 0,C 180,E1 -581.766,E2 -581.766} C_VEL
LIN {X 0,Y 601.426,Z 325.198,A -85,B 0,C 180,E1 -584.536,E2 -584.536} C_VEL
LIN {X 0,Y 601.38,Z 325.194,A -85,B 0,C 180,E1 -587.327,E2 -587.327} C_VEL
LIN {X 0,Y 601.401,Z 325.193,A -85,B 0,C 180,E1 -590.005,E2 -590.005} C_VEL
LIN {X 0,Y 601.432,Z 325.196,A -85,B 0,C 180,E1 -592.619,E2 -592.619} C_VEL
LIN {X 0,Y 601.386,Z 325.195,A -85,B 0,C 180,E1 -595.067,E2 -595.067} C_VEL
LIN {X 0,Y 601.407,Z 325.19,A -85,B 0,C 180,E1 -597.483,E2 -597.483} C_VEL
LIN {X 0,Y 601.409,Z 325.191,A -85,B 0,C 180,E1 -599.856,E2 -599.856} C_VEL
LIN {X 0,Y 601.402,Z 325.198,A -85,B 0,C 180,E1 -602.641,E2 -602.641} C_VEL
LIN {X 0,Y 601.387,Z 325.193,A -85,B 0,C 180,E1 -605.121,E2 -605.121} C_VEL
LIN {X 0,Y 601.398,Z 325.195,A -85,B 0,C 180,E1 -608.041,E2 -608.041} C_VEL
LIN {X 0,Y 601.407,Z 325.193,A -85,B 0,C 180,E1 -610.901,E2 -610.901} C_VEL
LIN {X 0,Y 601.412,Z 325.19,A -85,B 0,C 180,E1 -613.713,E2 -613.713} C_VEL
LIN {X 0,Y 601.403,Z 325.199,A -85,B 0,C 180,E1 -616.484,E2 -616.484} C_VEL
LIN {X 0,Y 601.367,Z 325.195,A -85,B 0,C 180,E1 -619.223,E2 -619.223} C_VEL
LIN {X 0,Y 601.439,Z 325.19,A -85,B 0,C 180,E1 -621.94,E2 -621.94} C_VEL
LIN {X 0,Y 601.402,Z 325.195,A -85,B 0,C 180,E1 -624.636,E2 -624.636} C_VEL
LIN {X 0,Y 601.402,Z 325.19,A -85,B 0,C 180,E1 -627.321,E2 -627.321} C_VEL
LIN {X 0,Y 601.446,Z 325.191,A -85,B 0,C 180,E1 -630,E2 -630} C_VEL
LIN {X 0,Y 601.412,Z 325.193,A -85,B 0,C 180,E1 -632.679,E2 -632.679} C_VEL
LIN {X 0,Y 601.387,Z 325.193,A -85,B 0,C 180,E1 -635.365,E2 -635.365} C_VEL
LIN {X 0,Y 601.431,Z 325.195,A -85,B 0,C 180,E1 -638.061,E2 -638.061} C_VEL
LIN {X 0,Y 601.366,Z 325.197,A -85,B 0,C 180,E1 -640.777,E2 -640.777} C_VEL
LIN {X 0,Y 601.383,Z 325.194,A -85,B 0,C 180,E1 -643.517,E2 -643.517} C_VEL
LIN {X 0,Y 601.41,Z 325.199,A -85,B 0,C 180,E1 -646.288,E2 -646.288} C_VEL
LIN {X 0,Y 601.378,Z 325.331,A -85,B 0,C 180,E1 -649.211,E2 -649.211} C_VEL
LIN {X 0,Y 601.535,Z 333.163,A -85,B 0,C 180,E1 -650.34,E2 -650.34} C_VEL
LIN {X 0,Y 601.504,Z 340.409,A -85,B 0,C 180,E1 -651.371,E2 -651.371} C_VEL
LIN {X 0,Y 602.024,Z 343.662,A -85,B 0,C 180,E1 -651.441,E2 -651.441} C_VEL
LIN {X 0,Y 601.859,Z 505.346,A -85,B 0,C 180,E1 -653.438,E2 -653.438} C_VEL
LIN {X 0,Y 601.836,Z 521.165,A -85,B 0,C 180,E1 -653.781,E2 -653.781} C_VEL
LIN {X 0,Y 601.782,Z 535.945,A -85,B 0,C 180,E1 -654.242,E2 -654.242} C_VEL
LIN {X 0,Y 601.69,Z 551.031,A -85,B 0,C 180,E1 -654.866,E2 -654.866} C_VEL
LIN {X 0,Y 601.636,Z 565.169,A -85,B 0,C 180,E1 -655.608,E2 -655.608} C_VEL
LIN {X 0,Y 601.578,Z 578.235,A -85,B 0,C 180,E1 -656.449,E2 -656.449} C_VEL
LIN {X 0,Y 601.53,Z 590.291,A -85,B 0,C 180,E1 -657.383,E2 -657.383} C_VEL
LIN {X 0,Y 601.463,Z 601.69,A -85,B 0,C 180,E1 -658.435,E2 -658.435} C_VEL
LIN {X 0,Y 601.456,Z 612.09,A -85,B 0,C 180,E1 -659.584,E2 -659.584} C_VEL
LIN {X 0,Y 601.407,Z 620.949,A -85,B 0,C 180,E1 -660.748,E2 -660.748} C_VEL
LIN {X 0,Y 601.378,Z 629.546,A -85,B 0,C 180,E1 -662.123,E2 -662.123} C_VEL
LIN {X 0,Y 601.367,Z 635.627,A -85,B 0,C 180,E1 -663.318,E2 -663.318} C_VEL
LIN {X 0,Y 601.341,Z 640.608,A -85,B 0,C 180,E1 -664.53,E2 -664.53} C_VEL
LIN {X 0,Y 601.34,Z 644.585,A -85,B 0,C 180,E1 -665.758,E2 -665.758} C_VEL
LIN {X 0,Y 601.328,Z 646.658,A -85,B 0,C 180,E1 -666.589,E2 -666.589} C_VEL
LIN {X 0,Y 601.331,Z 648.286,A -85,B 0,C 180,E1 -667.427,E2 -667.427} C_VEL
LIN {X 0,Y 601.314,Z 649.682,A -85,B 0,C 180,E1 -668.456,E2 -668.456} C_VEL
LIN {X 0,Y 601.303,Z 650.496,A -85,B 0,C 180,E1 -670.004,E2 -670.004} C_VEL
LIN {X 0,Y 601.321,Z 649.743,A -85,B 0,C 180,E1 -671.581,E2 -671.581} C_VEL
LIN {X 0,Y 601.341,Z 648.263,A -85,B 0,C 180,E1 -672.677,E2 -672.677} C_VEL
LIN {X 0,Y 601.332,Z 645.306,A -85,B 0,C 180,E1 -674.059,E2 -674.059} C_VEL
LIN {X 0,Y 601.34,Z 640.927,A -85,B 0,C 180,E1 -675.473,E2 -675.473} C_VEL
LIN {X 0,Y 601.368,Z 635.101,A -85,B 0,C 180,E1 -676.882,E2 -676.882} C_VEL
LIN {X 0,Y 601.383,Z 628.011,A -85,B 0,C 180,E1 -678.231,E2 -678.231} C_VEL
LIN {X 0,Y 601.404,Z 620.331,A -85,B 0,C 180,E1 -679.428,E2 -679.428} C_VEL
LIN {X 0,Y 601.451,Z 610.69,A -85,B 0,C 180,E1 -680.672,E2 -680.672} C_VEL
LIN {X 0,Y 601.49,Z 599.754,A -85,B 0,C 180,E1 -681.843,E2 -681.843} C_VEL
LIN {X 0,Y 601.532,Z 587.817,A -85,B 0,C 180,E1 -682.908,E2 -682.908} C_VEL
LIN {X 0,Y 601.624,Z 576.043,A -85,B 0,C 180,E1 -683.789,E2 -683.789} C_VEL
LIN {X 0,Y 601.655,Z 563.069,A -85,B 0,C 180,E1 -684.599,E2 -684.599} C_VEL
LIN {X 0,Y 601.711,Z 549.532,A -85,B 0,C 180,E1 -685.291,E2 -685.291} C_VEL
LIN {X 0,Y 601.779,Z 535.78,A -85,B 0,C 180,E1 -685.853,E2 -685.853} C_VEL
LIN {X 0,Y 601.842,Z 520.545,A -85,B 0,C 180,E1 -686.325,E2 -686.325} C_VEL
LIN {X 0,Y 601.872,Z 505.342,A -85,B 0,C 180,E1 -686.652,E2 -686.652} C_VEL
LIN {X 0,Y 601.962,Z 342.592,A -85,B 0,C 180,E1 -688.664,E2 -688.664} C_VEL
LIN {X 0,Y 601.51,Z 340.382,A -85,B 0,C 180,E1 -688.723,E2 -688.723} C_VEL
LIN {X 0,Y 601.498,Z 325.971,A -85,B 0,C 180,E1 -690.782,E2 -690.782} C_VEL
LIN {X 0,Y 601.351,Z 325.201,A -85,B 0,C 180,E1 -690.946,E2 -690.946} C_VEL
LIN {X 0,Y 601.366,Z 325.202,A -85,B 0,C 180,E1 -693.634,E2 -693.634} C_VEL
LIN {X 0,Y 601.435,Z 325.197,A -85,B 0,C 180,E1 -695.858,E2 -695.858} C_VEL
LIN {X 0,Y 601.378,Z 325.194,A -85,B 0,C 180,E1 -698.759,E2 -698.759} C_VEL
LIN {X 0,Y 601.382,Z 325.2,A -85,B 0,C 180,E1 -701.607,E2 -701.607} C_VEL
LIN {X 0,Y 601.385,Z 325.194,A -85,B 0,C 180,E1 -704.408,E2 -704.408} C_VEL
LIN {X 0,Y 601.391,Z 325.193,A -85,B 0,C 180,E1 -706.483,E2 -706.483} C_VEL
LIN {X 0,Y 601.379,Z 325.197,A -85,B 0,C 180,E1 -709.223,E2 -709.223} C_VEL
LIN {X 0,Y 601.435,Z 325.192,A -85,B 0,C 180,E1 -711.939,E2 -711.939} C_VEL
LIN {X 0,Y 601.394,Z 325.192,A -85,B 0,C 180,E1 -714.635,E2 -714.635} C_VEL
LIN {X 0,Y 601.429,Z 325.193,A -85,B 0,C 180,E1 -717.321,E2 -717.321} C_VEL
LIN {X 0,Y 601.446,Z 325.189,A -85,B 0,C 180,E1 -720,E2 -720} C_VEL
LIN {X 0,Y 601.414,Z 325.189,A -85,B 0,C 180,E1 -722.679,E2 -722.679} C_VEL
LIN {X 0,Y 601.421,Z 325.197,A -85,B 0,C 180,E1 -725.364,E2 -725.364} C_VEL
LIN {X 0,Y 601.44,Z 325.188,A -85,B 0,C 180,E1 -728.061,E2 -728.061} C_VEL
LIN {X 0,Y 601.412,Z 325.193,A -85,B 0,C 180,E1 -731.004,E2 -731.004} C_VEL
LIN {X 0,Y 601.419,Z 325.196,A -85,B 0,C 180,E1 -733.516,E2 -733.516} C_VEL
LIN {X 0,Y 601.432,Z 325.187,A -85,B 0,C 180,E1 -736.287,E2 -736.287} C_VEL
LIN {X 0,Y 601.416,Z 325.196,A -85,B 0,C 180,E1 -739.099,E2 -739.099} C_VEL
LIN {X 0,Y 601.404,Z 325.191,A -85,B 0,C 180,E1 -741.959,E2 -741.959} C_VEL
LIN {X 0,Y 601.437,Z 325.186,A -85,B 0,C 180,E1 -744.292,E2 -744.292} C_VEL
LIN {X 0,Y 601.452,Z 325.194,A -85,B 0,C 180,E1 -747.111,E2 -747.111} C_VEL
LIN {X 0,Y 601.431,Z 325.187,A -85,B 0,C 180,E1 -750.148,E2 -750.148} C_VEL
LIN {X 0,Y 601.415,Z 325.193,A -85,B 0,C 180,E1 -752.714,E2 -752.714} C_VEL
LIN {X 0,Y 601.392,Z 325.202,A -85,B 0,C 180,E1 -755.111,E2 -755.111} C_VEL
LIN {X 0,Y 601.437,Z 325.19,A -85,B 0,C 180,E1 -757.419,E2 -757.419} C_VEL
LIN {X 0,Y 601.404,Z 325.191,A -85,B 0,C 180,E1 -759.996,E2 -759.996} C_VEL
LIN {X 0,Y 601.413,Z 325.195,A -85,B 0,C 180,E1 -762.67,E2 -762.67} C_VEL
LIN {X 0,Y 601.428,Z 325.19,A -85,B 0,C 180,E1 -765.482,E2 -765.482} C_VEL
LIN {X 0,Y 601.425,Z 325.191,A -85,B 0,C 180,E1 -768.407,E2 -768.407} C_VEL
LIN {X 0,Y 601.43,Z 325.198,A -85,B 0,C 180,E1 -770.875,E2 -770.875} C_VEL
LIN {X 0,Y 601.399,Z 325.193,A -85,B 0,C 180,E1 -773.416,E2 -773.416} C_VEL
LIN {X 0,Y 601.433,Z 325.188,A -85,B 0,C 180,E1 -776.064,E2 -776.064} C_VEL
LIN {X 0,Y 601.412,Z 325.195,A -85,B 0,C 180,E1 -779.057,E2 -779.057} C_VEL
LIN {X 0,Y 601.412,Z 325.192,A -85,B 0,C 180,E1 -781.372,E2 -781.372} C_VEL
LIN {X 0,Y 601.414,Z 325.234,A -85,B 0,C 180,E1 -783.333,E2 -783.333} C_VEL
LIN {X 0,Y 601.978,Z 327.941,A -85,B 0,C 180,E1 -783.663,E2 -783.663} C_VEL
LIN {X 0,Y 601.86,Z 352.932,A -85,B 0,C 180,E1 -786.425,E2 -786.425} C_VEL
LIN {X 0,Y 601.731,Z 380.167,A -85,B 0,C 180,E1 -789.372,E2 -789.372} C_VEL
LIN {X 0,Y 601.644,Z 398.447,A -85,B 0,C 180,E1 -791.318,E2 -791.318} C_VEL
LIN {X 0,Y 602.045,Z 402.926,A -85,B 0,C 180,E1 -791.388,E2 -791.388} C_VEL
LIN {X 0,Y 601.882,Z 564.38,A -85,B 0,C 180,E1 -793.378,E2 -793.378} C_VEL
LIN {X 0,Y 601.844,Z 579.881,A -85,B 0,C 180,E1 -793.704,E2 -793.704} C_VEL
LIN {X 0,Y 601.786,Z 594.783,A -85,B 0,C 180,E1 -794.158,E2 -794.158} C_VEL
LIN {X 0,Y 601.72,Z 609.753,A -85,B 0,C 180,E1 -794.764,E2 -794.764} C_VEL
LIN {X 0,Y 601.658,Z 623.228,A -85,B 0,C 180,E1 -795.455,E2 -795.455} C_VEL
LIN {X 0,Y 601.617,Z 636.446,A -85,B 0,C 180,E1 -796.283,E2 -796.283} C_VEL
LIN {X 0,Y 601.531,Z 648.281,A -85,B 0,C 180,E1 -797.174,E2 -797.174} C_VEL
LIN {X 0,Y 601.489,Z 659.745,A -85,B 0,C 180,E1 -798.201,E2 -798.201} C_VEL
LIN {X 0,Y 601.43,Z 669.386,A -85,B 0,C 180,E1 -799.224,E2 -799.224} C_VEL
LIN {X 0,Y 601.428,Z 678.852,A -85,B 0,C 180,E1 -800.414,E2 -800.414} C_VEL
LIN {X 0,Y 601.369,Z 686.728,A -85,B 0,C 180,E1 -801.6,E2 -801.6} C_VEL
LIN {X 0,Y 601.368,Z 694.086,A -85,B 0,C 180,E1 -802.951,E2 -802.951} C_VEL
LIN {X 0,Y 601.373,Z 699.923,A -85,B 0,C 180,E1 -804.299,E2 -804.299} C_VEL
LIN {X 0,Y 601.33,Z 703.382,A -85,B 0,C 180,E1 -805.307,E2 -805.307} C_VEL
LIN {X 0,Y 601.337,Z 706.886,A -85,B 0,C 180,E1 -806.65,E2 -806.65} C_VEL
LIN {X 0,Y 601.342,Z 709.192,A -85,B 0,C 180,E1 -807.99,E2 -807.99} C_VEL
LIN {X 0,Y 601.335,Z 710.35,A -85,B 0,C 180,E1 -809.33,E2 -809.33} C_VEL
LIN {X 0,Y 601.335,Z 710.35,A -85,B 0,C 180,E1 -810.669,E2 -810.669} C_VEL
LIN {X 0,Y 601.342,Z 709.192,A -85,B 0,C 180,E1 -812.009,E2 -812.009} C_VEL
LIN {X 0,Y 601.337,Z 706.886,A -85,B 0,C 180,E1 -813.35,E2 -813.35} C_VEL
LIN {X 0,Y 601.329,Z 703.384,A -85,B 0,C 180,E1 -814.692,E2 -814.692} C_VEL
LIN {X 0,Y 601.356,Z 698.609,A -85,B 0,C 180,E1 -816.037,E2 -816.037} C_VEL
LIN {X 0,Y 601.365,Z 692.427,A -85,B 0,C 180,E1 -817.386,E2 -817.386} C_VEL
LIN {X 0,Y 601.386,Z 684.655,A -85,B 0,C 180,E1 -818.738,E2 -818.738} C_VEL
LIN {X 0,Y 601.428,Z 676.372,A -85,B 0,C 180,E1 -819.925,E2 -819.925} C_VEL
LIN {X 0,Y 601.46,Z 665.934,A -85,B 0,C 180,E1 -821.164,E2 -821.164} C_VEL
LIN {X 0,Y 601.514,Z 656.195,A -85,B 0,C 180,E1 -822.14,E2 -822.14} C_VEL
LIN {X 0,Y 601.57,Z 644.02,A -85,B 0,C 180,E1 -823.168,E2 -823.168} C_VEL
LIN {X 0,Y 601.605,Z 632.082,A -85,B 0,C 180,E1 -824.011,E2 -824.011} C_VEL
LIN {X 0,Y 601.65,Z 618.533,A -85,B 0,C 180,E1 -824.804,E2 -824.804} C_VEL
LIN {X 0,Y 601.763,Z 603.85,A -85,B 0,C 180,E1 -825.495,E2 -825.495} C_VEL
LIN {X 0,Y 601.785,Z 589.627,A -85,B 0,C 180,E1 -826.016,E2 -826.016} C_VEL
LIN {X 0,Y 601.85,Z 574.747,A -85,B 0,C 180,E1 -826.419,E2 -826.419} C_VEL
LIN {X 0,Y 601.864,Z 559.793,A -85,B 0,C 180,E1 -826.689,E2 -826.689} C_VEL
LIN {X 0,Y 601.928,Z 399.939,A -85,B 0,C 180,E1 -828.653,E2 -828.653} C_VEL
LIN {X 0,Y 601.665,Z 398.316,A -85,B 0,C 180,E1 -828.695,E2 -828.695} C_VEL
LIN {X 0,Y 601.747,Z 372.931,A -85,B 0,C 180,E1 -831.406,E2 -831.406} C_VEL
LIN {X 0,Y 601.893,Z 346.731,A -85,B 0,C 180,E1 -834.254,E2 -834.254} C_VEL
LIN {X 0,Y 601.977,Z 327.947,A -85,B 0,C 180,E1 -836.336,E2 -836.336} C_VEL
LIN {X 0,Y 601.39,Z 325.198,A -85,B 0,C 180,E1 -836.691,E2 -836.691} C_VEL
LIN {X 0,Y 601.406,Z 325.201,A -85,B 0,C 180,E1 -839.393,E2 -839.393} C_VEL
LIN {X 0,Y 601.402,Z 325.195,A -85,B 0,C 180,E1 -841.726,E2 -841.726} C_VEL
LIN {X 0,Y 601.425,Z 325.188,A -85,B 0,C 180,E1 -844.118,E2 -844.118} C_VEL
LIN {X 0,Y 601.398,Z 325.192,A -85,B 0,C 180,E1 -846.583,E2 -846.583} C_VEL
LIN {X 0,Y 601.437,Z 325.192,A -85,B 0,C 180,E1 -849.535,E2 -849.535} C_VEL
LIN {X 0,Y 601.405,Z 325.191,A -85,B 0,C 180,E1 -852.59,E2 -852.59} C_VEL
LIN {X 0,Y 601.422,Z 325.189,A -85,B 0,C 180,E1 -854.535,E2 -854.535} C_VEL
LIN {X 0,Y 601.41,Z 325.197,A -85,B 0,C 180,E1 -857.409,E2 -857.409} C_VEL
LIN {X 0,Y 601.402,Z 325.191,A -85,B 0,C 180,E1 -860.004,E2 -860.004} C_VEL
LIN {X 0,Y 601.431,Z 325.189,A -85,B 0,C 180,E1 -862.618,E2 -862.618} C_VEL
LIN {X 0,Y 601.439,Z 325.195,A -85,B 0,C 180,E1 -865.07,E2 -865.07} C_VEL
LIN {X 0,Y 601.427,Z 325.192,A -85,B 0,C 180,E1 -867.484,E2 -867.484} C_VEL
LIN {X 0,Y 601.426,Z 325.188,A -85,B 0,C 180,E1 -869.851,E2 -869.851} C_VEL
LIN {X 0,Y 601.413,Z 325.192,A -85,B 0,C 180,E1 -872.637,E2 -872.637} C_VEL
LIN {X 0,Y 601.4,Z 325.201,A -85,B 0,C 180,E1 -875.122,E2 -875.122} C_VEL
LIN {X 0,Y 601.412,Z 325.194,A -85,B 0,C 180,E1 -877.394,E2 -877.394} C_VEL
LIN {X 0,Y 601.401,Z 325.191,A -85,B 0,C 180,E1 -880.191,E2 -880.191} C_VEL
LIN {X 0,Y 601.428,Z 325.198,A -85,B 0,C 180,E1 -883.014,E2 -883.014} C_VEL
LIN {X 0,Y 601.42,Z 325.188,A -85,B 0,C 180,E1 -885.908,E2 -885.908} C_VEL
LIN {X 0,Y 601.434,Z 325.19,A -85,B 0,C 180,E1 -888.542,E2 -888.542} C_VEL
LIN {X 0,Y 601.41,Z 325.195,A -85,B 0,C 180,E1 -891.262,E2 -891.262} C_VEL
LIN {X 0,Y 601.433,Z 325.187,A -85,B 0,C 180,E1 -893.963,E2 -893.963} C_VEL
LIN {X 0,Y 601.431,Z 325.193,A -85,B 0,C 180,E1 -896.651,E2 -896.651} C_VEL
LIN {X 0,Y 601.441,Z 325.189,A -85,B 0,C 180,E1 -899.331,E2 -899.331} C_VEL
LIN {X 0,Y 601.435,Z 325.187,A -85,B 0,C 180,E1 -902.009,E2 -902.009} C_VEL
LIN {X 0,Y 601.42,Z 325.196,A -85,B 0,C 180,E1 -904.692,E2 -904.692} C_VEL
LIN {X 0,Y 601.435,Z 325.189,A -85,B 0,C 180,E1 -907.385,E2 -907.385} C_VEL
LIN {X 0,Y 601.433,Z 325.187,A -85,B 0,C 180,E1 -910.095,E2 -910.095} C_VEL
LIN {X 0,Y 601.408,Z 325.193,A -85,B 0,C 180,E1 -912.376,E2 -912.376} C_VEL
LIN {X 0,Y 600.74,Z 325.283,A -85,B 0,C 180,E1 -912.935,E2 -912.935} C_VEL
LIN {X 0,Y 597.889,Z 325.64,A -85,B 0,C 180,E1 -913.843,E2 -913.843} C_VEL
LIN {X 0,Y 595.479,Z 325.937,A -85,B 0,C 180,E1 -914.573,E2 -914.573} C_VEL
LIN {X 0,Y 594.442,Z 326.063,A -85,B 0,C 180,E1 -915.137,E2 -915.137} C_VEL
LIN {X 0,Y 594.356,Z 326.071,A -85,B 0,C 180,E1 -915.328,E2 -915.328} C_VEL
LIN {X 0,Y 594.386,Z 326.068,A -85,B 0,C 180,E1 -917.194,E2 -917.194} C_VEL
LIN {X 0,Y 594.372,Z 326.067,A -85,B 0,C 180,E1 -920.054,E2 -920.054} C_VEL
LIN {X 0,Y 594.356,Z 326.075,A -85,B 0,C 180,E1 -922.968,E2 -922.968} C_VEL
LIN {X 0,Y 594.36,Z 326.071,A -85,B 0,C 180,E1 -925.194,E2 -925.194} C_VEL
LIN {X 0,Y 594.346,Z 326.07,A -85,B 0,C 180,E1 -927.52,E2 -927.52} C_VEL
LIN {X 0,Y 594.385,Z 326.069,A -85,B 0,C 180,E1 -930.329,E2 -930.329} C_VEL
LIN {X 0,Y 594.376,Z 326.072,A -85,B 0,C 180,E1 -932.951,E2 -932.951} C_VEL
LIN {X 0,Y 594.353,Z 326.069,A -85,B 0,C 180,E1 -935.409,E2 -935.409} C_VEL
LIN {X 0,Y 594.385,Z 326.066,A -85,B 0,C 180,E1 -937.941,E2 -937.941} C_VEL
LIN {X 0,Y 594.369,Z 326.073,A -85,B 0,C 180,E1 -940.822,E2 -940.822} C_VEL
LIN {X 0,Y 594.35,Z 326.07,A -85,B 0,C 180,E1 -943.301,E2 -943.301} C_VEL
LIN {X 0,Y 594.361,Z 326.071,A -85,B 0,C 180,E1 -946.162,E2 -946.162} C_VEL
LIN {X 0,Y 594.38,Z 326.076,A -85,B 0,C 180,E1 -948.537,E2 -948.537} C_VEL
LIN {X 0,Y 594.368,Z 326.067,A -85,B 0,C 180,E1 -951.298,E2 -951.298} C_VEL
LIN {X 0,Y 594.348,Z 326.07,A -85,B 0,C 180,E1 -953.756,E2 -953.756} C_VEL
LIN {X 0,Y 594.38,Z 326.071,A -85,B 0,C 180,E1 -956.239,E2 -956.239} C_VEL
LIN {X 0,Y 594.365,Z 326.075,A -85,B 0,C 180,E1 -958.65,E2 -958.65} C_VEL
LIN {X 0,Y 594.375,Z 326.068,A -85,B 0,C 180,E1 -961.045,E2 -961.045} C_VEL
LIN {X 0,Y 594.36,Z 326.068,A -85,B 0,C 180,E1 -963.3,E2 -963.3} C_VEL
LIN {X 0,Y 594.357,Z 326.068,A -85,B 0,C 180,E1 -965.574,E2 -965.574} C_VEL
LIN {X 0,Y 594.355,Z 326.078,A -85,B 0,C 180,E1 -968.497,E2 -968.497} C_VEL
LIN {X 0,Y 594.355,Z 326.068,A -85,B 0,C 180,E1 -971.382,E2 -971.382} C_VEL
LIN {X 0,Y 594.35,Z 326.077,A -85,B 0,C 180,E1 -974.219,E2 -974.219} C_VEL
LIN {X 0,Y 594.373,Z 326.076,A -85,B 0,C 180,E1 -976.321,E2 -976.321} C_VEL
LIN {X 0,Y 594.347,Z 326.07,A -85,B 0,C 180,E1 -979.094,E2 -979.094} C_VEL
LIN {X 0,Y 594.381,Z 326.068,A -85,B 0,C 180,E1 -981.843,E2 -981.843} C_VEL
LIN {X 0,Y 594.371,Z 326.072,A -85,B 0,C 180,E1 -984.572,E2 -984.572} C_VEL
LIN {X 0,Y 594.371,Z 326.066,A -85,B 0,C 180,E1 -987.289,E2 -987.289} C_VEL
LIN {X 0,Y 594.414,Z 326.067,A -85,B 0,C 180,E1 -990,E2 -990} C_VEL
LIN {X 0,Y 594.378,Z 326.069,A -85,B 0,C 180,E1 -992.711,E2 -992.711} C_VEL
LIN {X 0,Y 594.357,Z 326.069,A -85,B 0,C 180,E1 -995.428,E2 -995.428} C_VEL
LIN {X 0,Y 594.375,Z 326.076,A -85,B 0,C 180,E1 -998.158,E2 -998.158} C_VEL
LIN {X 0,Y 594.335,Z 326.071,A -85,B 0,C 180,E1 -1001.044,E2 -1001.044} C_VEL
LIN {X 0,Y 594.36,Z 326.071,A -85,B 0,C 180,E1 -1003.68,E2 -1003.68} C_VEL
LIN {X 0,Y 594.336,Z 326.074,A -85,B 0,C 180,E1 -1006.699,E2 -1006.699} C_VEL
LIN {X 0,Y 594.349,Z 326.187,A -85,B 0,C 180,E1 -1009.078,E2 -1009.078} C_VEL
LIN {X 0,Y 594.628,Z 331.532,A -85,B 0,C 180,E1 -1009.865,E2 -1009.865} C_VEL
LIN {X 0,Y 594.545,Z 340.498,A -85,B 0,C 180,E1 -1011.157,E2 -1011.157} C_VEL
LIN {X 0,Y 595.292,Z 344.387,A -85,B 0,C 180,E1 -1011.232,E2 -1011.232} C_VEL
LIN {X 0,Y 595.056,Z 505.063,A -85,B 0,C 180,E1 -1013.238,E2 -1013.238} C_VEL
LIN {X 0,Y 595.022,Z 521.004,A -85,B 0,C 180,E1 -1013.585,E2 -1013.585} C_VEL
LIN {X 0,Y 594.933,Z 535.822,A -85,B 0,C 180,E1 -1014.051,E2 -1014.051} C_VEL
LIN {X 0,Y 594.83,Z 550.217,A -85,B 0,C 180,E1 -1014.649,E2 -1014.649} C_VEL
LIN {X 0,Y 594.708,Z 563.932,A -85,B 0,C 180,E1 -1015.365,E2 -1015.365} C_VEL
LIN {X 0,Y 594.632,Z 577.584,A -85,B 0,C 180,E1 -1016.242,E2 -1016.242} C_VEL
LIN {X 0,Y 594.553,Z 590.64,A -85,B 0,C 180,E1 -1017.262,E2 -1017.262} C_VEL
LIN {X 0,Y 594.459,Z 600.959,A -85,B 0,C 180,E1 -1018.223,E2 -1018.223} C_VEL
LIN {X 0,Y 594.42,Z 611.49,A -85,B 0,C 180,E1 -1019.385,E2 -1019.385} C_VEL
LIN {X 0,Y 594.331,Z 620.427,A -85,B 0,C 180,E1 -1020.563,E2 -1020.563} C_VEL
LIN {X 0,Y 594.311,Z 628.613,A -85,B 0,C 180,E1 -1021.864,E2 -1021.864} C_VEL
LIN {X 0,Y 594.268,Z 634.305,A -85,B 0,C 180,E1 -1022.957,E2 -1022.957} C_VEL
LIN {X 0,Y 594.266,Z 639.364,A -85,B 0,C 180,E1 -1024.121,E2 -1024.121} C_VEL
LIN {X 0,Y 594.235,Z 643.76,A -85,B 0,C 180,E1 -1025.417,E2 -1025.417} C_VEL
LIN {X 0,Y 594.223,Z 646.477,A -85,B 0,C 180,E1 -1026.461,E2 -1026.461} C_VEL
LIN {X 0,Y 594.218,Z 649.125,A -85,B 0,C 180,E1 -1027.954,E2 -1027.954} C_VEL
LIN {X 0,Y 594.207,Z 650.002,A -85,B 0,C 180,E1 -1028.819,E2 -1028.819} C_VEL
LIN {X 0,Y 594.223,Z 650.44,A -85,B 0,C 180,E1 -1029.756,E2 -1029.756} C_VEL
LIN {X 0,Y 594.217,Z 650.321,A -85,B 0,C 180,E1 -1030.803,E2 -1030.803} C_VEL
LIN {X 0,Y 594.252,Z 648.788,A -85,B 0,C 180,E1 -1032.386,E2 -1032.386} C_VEL
LIN {X 0,Y 594.244,Z 646.039,A -85,B 0,C 180,E1 -1033.826,E2 -1033.826} C_VEL
LIN {X 0,Y 594.265,Z 642.113,A -85,B 0,C 180,E1 -1035.201,E2 -1035.201} C_VEL
LIN {X 0,Y 594.301,Z 636.356,A -85,B 0,C 180,E1 -1036.694,E2 -1036.694} C_VEL
LIN {X 0,Y 594.288,Z 630.338,A -85,B 0,C 180,E1 -1037.913,E2 -1037.913} C_VEL
LIN {X 0,Y 594.321,Z 622.718,A -85,B 0,C 180,E1 -1039.185,E2 -1039.185} C_VEL
LIN {X 0,Y 594.396,Z 614.551,A -85,B 0,C 180,E1 -1040.321,E2 -1040.321} C_VEL
LIN {X 0,Y 594.45,Z 604.802,A -85,B 0,C 180,E1 -1041.463,E2 -1041.463} C_VEL
LIN {X 0,Y 594.511,Z 593.874,A -85,B 0,C 180,E1 -1042.54,E2 -1042.54} C_VEL
LIN {X 0,Y 594.604,Z 582.435,A -85,B 0,C 180,E1 -1043.489,E2 -1043.489} C_VEL
LIN {X 0,Y 594.695,Z 569.167,A -85,B 0,C 180,E1 -1044.406,E2 -1044.406} C_VEL
LIN {X 0,Y 594.795,Z 555.31,A -85,B 0,C 180,E1 -1045.19,E2 -1045.19} C_VEL
LIN {X 0,Y 594.917,Z 541.066,A -85,B 0,C 180,E1 -1045.835,E2 -1045.835} C_VEL
LIN {X 0,Y 594.975,Z 526.498,A -85,B 0,C 180,E1 -1046.347,E2 -1046.347} C_VEL
LIN {X 0,Y 595.039,Z 510.964,A -85,B 0,C 180,E1 -1046.74,E2 -1046.74} C_VEL
LIN {X 0,Y 595.089,Z 494.063,A -85,B 0,C 180,E1 -1047.005,E2 -1047.005} C_VEL
LIN {X 0,Y 595.198,Z 343.6,A -85,B 0,C 180,E1 -1048.871,E2 -1048.871} C_VEL
LIN {X 0,Y 594.533,Z 340.431,A -85,B 0,C 180,E1 -1048.943,E2 -1048.943} C_VEL
LIN {X 0,Y 594.574,Z 327.464,A -85,B 0,C 180,E1 -1050.818,E2 -1050.818} C_VEL
LIN {X 0,Y 594.33,Z 326.077,A -85,B 0,C 180,E1 -1051.052,E2 -1051.052} C_VEL
LIN {X 0,Y 594.335,Z 326.081,A -85,B 0,C 180,E1 -1053.988,E2 -1053.988} C_VEL
LIN {X 0,Y 594.354,Z 326.073,A -85,B 0,C 180,E1 -1056.294,E2 -1056.294} C_VEL
LIN {X 0,Y 594.378,Z 326.067,A -85,B 0,C 180,E1 -1059.223,E2 -1059.223} C_VEL
LIN {X 0,Y 594.328,Z 326.077,A -85,B 0,C 180,E1 -1062.094,E2 -1062.094} C_VEL
LIN {X 0,Y 594.341,Z 326.074,A -85,B 0,C 180,E1 -1064.218,E2 -1064.218} C_VEL
LIN {X 0,Y 594.364,Z 326.07,A -85,B 0,C 180,E1 -1066.32,E2 -1066.32} C_VEL
LIN {X 0,Y 594.366,Z 326.069,A -85,B 0,C 180,E1 -1069.094,E2 -1069.094} C_VEL
LIN {X 0,Y 594.379,Z 326.073,A -85,B 0,C 180,E1 -1071.843,E2 -1071.843} C_VEL
LIN {X 0,Y 594.363,Z 326.068,A -85,B 0,C 180,E1 -1074.572,E2 -1074.572} C_VEL
LIN {X 0,Y 594.394,Z 326.069,A -85,B 0,C 180,E1 -1077.289,E2 -1077.289} C_VEL
LIN {X 0,Y 594.415,Z 326.065,A -85,B 0,C 180,E1 -1080,E2 -1080} C_VEL
LIN {X 0,Y 594.384,Z 326.065,A -85,B 0,C 180,E1 -1082.711,E2 -1082.711} C_VEL
LIN {X 0,Y 594.387,Z 326.074,A -85,B 0,C 180,E1 -1085.428,E2 -1085.428} C_VEL
LIN {X 0,Y 594.383,Z 326.066,A -85,B 0,C 180,E1 -1088.157,E2 -1088.157} C_VEL
LIN {X 0,Y 594.378,Z 326.071,A -85,B 0,C 180,E1 -1091.066,E2 -1091.066} C_VEL
LIN {X 0,Y 594.383,Z 326.07,A -85,B 0,C 180,E1 -1093.679,E2 -1093.679} C_VEL
LIN {X 0,Y 594.369,Z 326.068,A -85,B 0,C 180,E1 -1096.71,E2 -1096.71} C_VEL
LIN {X 0,Y 594.367,Z 326.077,A -85,B 0,C 180,E1 -1099.334,E2 -1099.334} C_VEL
LIN {X 0,Y 594.362,Z 326.074,A -85,B 0,C 180,E1 -1101.503,E2 -1101.503} C_VEL
LIN {X 0,Y 594.391,Z 326.064,A -85,B 0,C 180,E1 -1104.446,E2 -1104.446} C_VEL
LIN {X 0,Y 594.383,Z 326.068,A -85,B 0,C 180,E1 -1106.699,E2 -1106.699} C_VEL
LIN {X 0,Y 594.381,Z 326.074,A -85,B 0,C 180,E1 -1108.998,E2 -1108.998} C_VEL
LIN {X 0,Y 594.378,Z 326.068,A -85,B 0,C 180,E1 -1111.642,E2 -1111.642} C_VEL
LIN {X 0,Y 594.378,Z 326.069,A -85,B 0,C 180,E1 -1114.58,E2 -1114.58} C_VEL
LIN {X 0,Y 594.392,Z 326.066,A -85,B 0,C 180,E1 -1117.608,E2 -1117.608} C_VEL
LIN {X 0,Y 594.371,Z 326.071,A -85,B 0,C 180,E1 -1120.567,E2 -1120.567} C_VEL
LIN {X 0,Y 594.368,Z 326.072,A -85,B 0,C 180,E1 -1123.299,E2 -1123.299} C_VEL
LIN {X 0,Y 594.384,Z 326.066,A -85,B 0,C 180,E1 -1126.159,E2 -1126.159} C_VEL
LIN {X 0,Y 594.377,Z 326.071,A -85,B 0,C 180,E1 -1129.178,E2 -1129.178} C_VEL
LIN {X 0,Y 594.384,Z 326.066,A -85,B 0,C 180,E1 -1132.059,E2 -1132.059} C_VEL
LIN {X 0,Y 594.35,Z 326.078,A -85,B 0,C 180,E1 -1134.677,E2 -1134.677} C_VEL
LIN {X 0,Y 594.377,Z 326.071,A -85,B 0,C 180,E1 -1137.089,E2 -1137.089} C_VEL
LIN {X 0,Y 594.387,Z 326.066,A -85,B 0,C 180,E1 -1139.672,E2 -1139.672} C_VEL
LIN {X 0,Y 594.376,Z 326.077,A -85,B 0,C 180,E1 -1142.539,E2 -1142.539} C_VEL
LIN {X 0,Y 594.414,Z 326.275,A -85,B 0,C 180,E1 -1143.112,E2 -1143.112} C_VEL
LIN {X 0,Y 595.23,Z 330.915,A -85,B 0,C 180,E1 -1143.678,E2 -1143.678} C_VEL
LIN {X 0,Y 595.052,Z 356.264,A -85,B 0,C 180,E1 -1146.508,E2 -1146.508} C_VEL
LIN {X 0,Y 594.86,Z 382.922,A -85,B 0,C 180,E1 -1149.422,E2 -1149.422} C_VEL
LIN {X 0,Y 594.74,Z 398.455,A -85,B 0,C 180,E1 -1151.094,E2 -1151.094} C_VEL
LIN {X 0,Y 595.33,Z 402.066,A -85,B 0,C 180,E1 -1151.159,E2 -1151.159} C_VEL
LIN {X 0,Y 595.071,Z 565.424,A -85,B 0,C 180,E1 -1153.2,E2 -1153.2} C_VEL
LIN {X 0,Y 595.007,Z 581.475,A -85,B 0,C 180,E1 -1153.554,E2 -1153.554} C_VEL
LIN {X 0,Y 594.933,Z 596.039,A -85,B 0,C 180,E1 -1154.014,E2 -1154.014} C_VEL
LIN {X 0,Y 594.858,Z 609.755,A -85,B 0,C 180,E1 -1154.584,E2 -1154.584} C_VEL
LIN {X 0,Y 594.732,Z 623.23,A -85,B 0,C 180,E1 -1155.281,E2 -1155.281} C_VEL
LIN {X 0,Y 594.681,Z 635.788,A -85,B 0,C 180,E1 -1156.075,E2 -1156.075} C_VEL
LIN {X 0,Y 594.56,Z 648.282,A -85,B 0,C 180,E1 -1157.021,E2 -1157.021} C_VEL
LIN {X 0,Y 594.466,Z 659.745,A -85,B 0,C 180,E1 -1158.059,E2 -1158.059} C_VEL
LIN {X 0,Y 594.388,Z 669.387,A -85,B 0,C 180,E1 -1159.095,E2 -1159.095} C_VEL
LIN {X 0,Y 594.367,Z 678.853,A -85,B 0,C 180,E1 -1160.299,E2 -1160.299} C_VEL
LIN {X 0,Y 594.311,Z 686.729,A -85,B 0,C 180,E1 -1161.499,E2 -1161.499} C_VEL
LIN {X 0,Y 594.292,Z 694.087,A -85,B 0,C 180,E1 -1162.867,E2 -1162.867} C_VEL
LIN {X 0,Y 594.298,Z 699.923,A -85,B 0,C 180,E1 -1164.231,E2 -1164.231} C_VEL
LIN {X 0,Y 594.232,Z 703.383,A -85,B 0,C 180,E1 -1165.251,E2 -1165.251} C_VEL
LIN {X 0,Y 594.257,Z 706.886,A -85,B 0,C 180,E1 -1166.61,E2 -1166.61} C_VEL
LIN {X 0,Y 594.241,Z 709.192,A -85,B 0,C 180,E1 -1167.966,E2 -1167.966} C_VEL
LIN {X 0,Y 594.235,Z 710.35,A -85,B 0,C 180,E1 -1169.322,E2 -1169.322} C_VEL
LIN {X 0,Y 594.235,Z 710.35,A -85,B 0,C 180,E1 -1170.677,E2 -1170.677} C_VEL
LIN {X 0,Y 594.241,Z 709.193,A -85,B 0,C 180,E1 -1172.033,E2 -1172.033} C_VEL
LIN {X 0,Y 594.257,Z 706.887,A -85,B 0,C 180,E1 -1173.39,E2 -1173.39} C_VEL
LIN {X 0,Y 594.232,Z 703.385,A -85,B 0,C 180,E1 -1174.749,E2 -1174.749} C_VEL
LIN {X 0,Y 594.278,Z 698.609,A -85,B 0,C 180,E1 -1176.11,E2 -1176.11} C_VEL
LIN {X 0,Y 594.287,Z 692.426,A -85,B 0,C 180,E1 -1177.474,E2 -1177.474} C_VEL
LIN {X 0,Y 594.33,Z 684.654,A -85,B 0,C 180,E1 -1178.843,E2 -1178.843} C_VEL
LIN {X 0,Y 594.388,Z 676.372,A -85,B 0,C 180,E1 -1180.044,E2 -1180.044} C_VEL
LIN {X 0,Y 594.433,Z 666.561,A -85,B 0,C 180,E1 -1181.231,E2 -1181.231} C_VEL
LIN {X 0,Y 594.53,Z 656.195,A -85,B 0,C 180,E1 -1182.285,E2 -1182.285} C_VEL
LIN {X 0,Y 594.581,Z 644.021,A -85,B 0,C 180,E1 -1183.326,E2 -1183.326} C_VEL
LIN {X 0,Y 594.693,Z 632.079,A -85,B 0,C 180,E1 -1184.177,E2 -1184.177} C_VEL
LIN {X 0,Y 594.75,Z 618.53,A -85,B 0,C 180,E1 -1184.98,E2 -1184.98} C_VEL
LIN {X 0,Y 594.903,Z 603.847,A -85,B 0,C 180,E1 -1185.678,E2 -1185.678} C_VEL
LIN {X 0,Y 594.966,Z 589.627,A -85,B 0,C 180,E1 -1186.204,E2 -1186.204} C_VEL
LIN {X 0,Y 595.04,Z 575.154,A -85,B 0,C 180,E1 -1186.602,E2 -1186.602} C_VEL
LIN {X 0,Y 595.064,Z 559.793,A -85,B 0,C 180,E1 -1186.885,E2 -1186.885} C_VEL
LIN {X 0,Y 595.235,Z 401.215,A -85,B 0,C 180,E1 -1188.855,E2 -1188.855} C_VEL
LIN {X 0,Y 594.74,Z 398.454,A -85,B 0,C 180,E1 -1188.906,E2 -1188.906} C_VEL
LIN {X 0,Y 594.888,Z 374.597,A -85,B 0,C 180,E1 -1191.483,E2 -1191.483} C_VEL
LIN {X 0,Y 595.067,Z 349.606,A -85,B 0,C 180,E1 -1194.23,E2 -1194.23} C_VEL
LIN {X 0,Y 595.227,Z 330.637,A -85,B 0,C 180,E1 -1196.353,E2 -1196.353} C_VEL
LIN {X 0,Y 594.375,Z 326.074,A -85,B 0,C 180,E1 -1196.937,E2 -1196.937} C_VEL
LIN {X 0,Y 594.372,Z 326.071,A -85,B 0,C 180,E1 -1199.776,E2 -1199.776} C_VEL
LIN {X 0,Y 594.358,Z 326.069,A -85,B 0,C 180,E1 -1202.147,E2 -1202.147} C_VEL
LIN {X 0,Y 594.372,Z 326.068,A -85,B 0,C 180,E1 -1204.58,E2 -1204.58} C_VEL
LIN {X 0,Y 594.388,Z 326.07,A -85,B 0,C 180,E1 -1207.608,E2 -1207.608} C_VEL
LIN {X 0,Y 594.365,Z 326.068,A -85,B 0,C 180,E1 -1210.567,E2 -1210.567} C_VEL
LIN {X 0,Y 594.377,Z 326.075,A -85,B 0,C 180,E1 -1213.298,E2 -1213.298} C_VEL
LIN {X 0,Y 594.364,Z 326.067,A -85,B 0,C 180,E1 -1216.16,E2 -1216.16} C_VEL
LIN {X 0,Y 594.383,Z 326.076,A -85,B 0,C 180,E1 -1219.177,E2 -1219.177} C_VEL
LIN {X 0,Y 594.384,Z 326.065,A -85,B 0,C 180,E1 -1222.059,E2 -1222.059} C_VEL
LIN {X 0,Y 594.382,Z 326.068,A -85,B 0,C 180,E1 -1224.672,E2 -1224.672} C_VEL
LIN {X 0,Y 594.375,Z 326.076,A -85,B 0,C 180,E1 -1227.088,E2 -1227.088} C_VEL
LIN {X 0,Y 594.384,Z 326.067,A -85,B 0,C 180,E1 -1229.672,E2 -1229.672} C_VEL
LIN {X 0,Y 594.371,Z 326.068,A -85,B 0,C 180,E1 -1232.539,E2 -1232.539} C_VEL
LIN {X 0,Y 594.372,Z 326.072,A -85,B 0,C 180,E1 -1234.807,E2 -1234.807} C_VEL
LIN {X 0,Y 594.362,Z 326.075,A -85,B 0,C 180,E1 -1237.265,E2 -1237.265} C_VEL
LIN {X 0,Y 594.371,Z 326.066,A -85,B 0,C 180,E1 -1239.946,E2 -1239.946} C_VEL
LIN {X 0,Y 594.387,Z 326.071,A -85,B 0,C 180,E1 -1242.807,E2 -1242.807} C_VEL
LIN {X 0,Y 594.387,Z 326.065,A -85,B 0,C 180,E1 -1245.826,E2 -1245.826} C_VEL
LIN {X 0,Y 594.393,Z 326.066,A -85,B 0,C 180,E1 -1248.404,E2 -1248.404} C_VEL
LIN {X 0,Y 594.377,Z 326.073,A -85,B 0,C 180,E1 -1251.158,E2 -1251.158} C_VEL
LIN {X 0,Y 594.382,Z 326.065,A -85,B 0,C 180,E1 -1253.891,E2 -1253.891} C_VEL
LIN {X 0,Y 594.382,Z 326.07,A -85,B 0,C 180,E1 -1256.611,E2 -1256.611} C_VEL
LIN {X 0,Y 594.413,Z 326.065,A -85,B 0,C 180,E1 -1259.323,E2 -1259.323} C_VEL
LIN {X 0,Y 594.403,Z 326.063,A -85,B 0,C 180,E1 -1262.033,E2 -1262.033} C_VEL
LIN {X 0,Y 594.389,Z 326.073,A -85,B 0,C 180,E1 -1264.748,E2 -1264.748} C_VEL
LIN {X 0,Y 594.39,Z 326.066,A -85,B 0,C 180,E1 -1267.473,E2 -1267.473} C_VEL
LIN {X 0,Y 594.393,Z 326.065,A -85,B 0,C 180,E1 -1270.216,E2 -1270.216} C_VEL
LIN {X 0,Y 594.363,Z 326.075,A -85,B 0,C 180,E1 -1272.983,E2 -1272.983} C_VEL
LIN {X 0,Y 594.356,Z 326.071,A -85,B 0,C 180,E1 -1275.328,E2 -1275.328} C_VEL
LIN {X 0,Y 593.682,Z 326.155,A -85,B 0,C 180,E1 -1275.893,E2 -1275.893} C_VEL
LIN {X 0,Y 590.817,Z 326.52,A -85,B 0,C 180,E1 -1276.812,E2 -1276.812} C_VEL
LIN {X 0,Y 588.408,Z 326.814,A -85,B 0,C 180,E1 -1277.55,E2 -1277.55} C_VEL
LIN {X 0,Y 587.386,Z 326.938,A -85,B 0,C 180,E1 -1278.12,E2 -1278.12} C_VEL
LIN {X 0,Y 587.309,Z 326.948,A -85,B 0,C 180,E1 -1278.313,E2 -1278.313} C_VEL
LIN {X 0,Y 587.329,Z 326.949,A -85,B 0,C 180,E1 -1281.038,E2 -1281.038} C_VEL
LIN {X 0,Y 587.314,Z 326.948,A -85,B 0,C 180,E1 -1283.259,E2 -1283.259} C_VEL
LIN {X 0,Y 587.323,Z 326.945,A -85,B 0,C 180,E1 -1285.518,E2 -1285.518} C_VEL
LIN {X 0,Y 587.306,Z 326.947,A -85,B 0,C 180,E1 -1287.82,E2 -1287.82} C_VEL
LIN {X 0,Y 587.334,Z 326.95,A -85,B 0,C 180,E1 -1290.51,E2 -1290.51} C_VEL
LIN {X 0,Y 587.327,Z 326.945,A -85,B 0,C 180,E1 -1293.398,E2 -1293.398} C_VEL
LIN {X 0,Y 587.317,Z 326.946,A -85,B 0,C 180,E1 -1295.899,E2 -1295.899} C_VEL
LIN {X 0,Y 587.327,Z 326.952,A -85,B 0,C 180,E1 -1298.48,E2 -1298.48} C_VEL
LIN {X 0,Y 587.331,Z 326.946,A -85,B 0,C 180,E1 -1301.158,E2 -1301.158} C_VEL
LIN {X 0,Y 587.303,Z 326.95,A -85,B 0,C 180,E1 -1304.111,E2 -1304.111} C_VEL
LIN {X 0,Y 587.297,Z 326.951,A -85,B 0,C 180,E1 -1306.992,E2 -1306.992} C_VEL
LIN {X 0,Y 587.308,Z 326.947,A -85,B 0,C 180,E1 -1309.746,E2 -1309.746} C_VEL
LIN {X 0,Y 587.342,Z 326.95,A -85,B 0,C 180,E1 -1312.393,E2 -1312.393} C_VEL
LIN {X 0,Y 587.355,Z 326.941,A -85,B 0,C 180,E1 -1315.78,E2 -1315.78} C_VEL
LIN {X 0,Y 587.333,Z 326.949,A -85,B 0,C 180,E1 -1318.231,E2 -1318.231} C_VEL
LIN {X 0,Y 587.344,Z 326.946,A -85,B 0,C 180,E1 -1320.869,E2 -1320.869} C_VEL
LIN {X 0,Y 587.311,Z 326.947,A -85,B 0,C 180,E1 -1323.83,E2 -1323.83} C_VEL
LIN {X 0,Y 587.305,Z 326.95,A -85,B 0,C 180,E1 -1325.993,E2 -1325.993} C_VEL
LIN {X 0,Y 587.335,Z 326.945,A -85,B 0,C 180,E1 -1328.963,E2 -1328.963} C_VEL
LIN {X 0,Y 587.288,Z 326.951,A -85,B 0,C 180,E1 -1331.872,E2 -1331.872} C_VEL
LIN {X 0,Y 587.307,Z 326.951,A -85,B 0,C 180,E1 -1334.737,E2 -1334.737} C_VEL
LIN {X 0,Y 587.282,Z 326.952,A -85,B 0,C 180,E1 -1336.858,E2 -1336.858} C_VEL
LIN {X 0,Y 587.326,Z 326.945,A -85,B 0,C 180,E1 -1339.66,E2 -1339.66} C_VEL
LIN {X 0,Y 587.317,Z 326.954,A -85,B 0,C 180,E1 -1342.437,E2 -1342.437} C_VEL
LIN {X 0,Y 587.33,Z 326.944,A -85,B 0,C 180,E1 -1345.195,E2 -1345.195} C_VEL
LIN {X 0,Y 587.37,Z 326.943,A -85,B 0,C 180,E1 -1347.943,E2 -1347.943} C_VEL
LIN {X 0,Y 587.37,Z 326.942,A -85,B 0,C 180,E1 -1350.686,E2 -1350.686} C_VEL
LIN {X 0,Y 587.345,Z 326.944,A -85,B 0,C 180,E1 -1352.744,E2 -1352.744} C_VEL
LIN {X 0,Y 587.326,Z 326.945,A -85,B 0,C 180,E1 -1355.494,E2 -1355.494} C_VEL
LIN {X 0,Y 587.334,Z 326.953,A -85,B 0,C 180,E1 -1358.256,E2 -1358.256} C_VEL
LIN {X 0,Y 587.302,Z 326.947,A -85,B 0,C 180,E1 -1361.107,E2 -1361.107} C_VEL
LIN {X 0,Y 587.346,Z 326.947,A -85,B 0,C 180,E1 -1363.846,E2 -1363.846} C_VEL
LIN {X 0,Y 587.288,Z 326.952,A -85,B 0,C 180,E1 -1366.793,E2 -1366.793} C_VEL
LIN {X 0,Y 587.313,Z 327,A -85,B 0,C 180,E1 -1368.935,E2 -1368.935} C_VEL
LIN {X 0,Y 587.678,Z 332.416,A -85,B 0,C 180,E1 -1369.746,E2 -1369.746} C_VEL
LIN {X 0,Y 587.593,Z 340.421,A -85,B 0,C 180,E1 -1370.913,E2 -1370.913} C_VEL
LIN {X 0,Y 588.537,Z 344.894,A -85,B 0,C 180,E1 -1371.014,E2 -1371.014} C_VEL
LIN {X 0,Y 588.274,Z 504.654,A -85,B 0,C 180,E1 -1373.032,E2 -1373.032} C_VEL
LIN {X 0,Y 588.205,Z 519.938,A -85,B 0,C 180,E1 -1373.362,E2 -1373.362} C_VEL
LIN {X 0,Y 588.085,Z 535.071,A -85,B 0,C 180,E1 -1373.834,E2 -1373.834} C_VEL
LIN {X 0,Y 587.987,Z 549.81,A -85,B 0,C 180,E1 -1374.447,E2 -1374.447} C_VEL
LIN {X 0,Y 587.82,Z 562.627,A -85,B 0,C 180,E1 -1375.115,E2 -1375.115} C_VEL
LIN {X 0,Y 587.702,Z 576.041,A -85,B 0,C 180,E1 -1375.969,E2 -1375.969} C_VEL
LIN {X 0,Y 587.577,Z 588.629,A -85,B 0,C 180,E1 -1376.938,E2 -1376.938} C_VEL
LIN {X 0,Y 587.45,Z 600.219,A -85,B 0,C 180,E1 -1378.007,E2 -1378.007} C_VEL
LIN {X 0,Y 587.365,Z 610.475,A -85,B 0,C 180,E1 -1379.135,E2 -1379.135} C_VEL
LIN {X 0,Y 587.29,Z 619.635,A -85,B 0,C 180,E1 -1380.336,E2 -1380.336} C_VEL
LIN {X 0,Y 587.244,Z 627.504,A -85,B 0,C 180,E1 -1381.574,E2 -1381.574} C_VEL
LIN {X 0,Y 587.185,Z 634.145,A -85,B 0,C 180,E1 -1382.837,E2 -1382.837} C_VEL
LIN {X 0,Y 587.164,Z 640.025,A -85,B 0,C 180,E1 -1384.233,E2 -1384.233} C_VEL
LIN {X 0,Y 587.152,Z 644.228,A -85,B 0,C 180,E1 -1385.517,E2 -1385.517} C_VEL
LIN {X 0,Y 587.126,Z 647.198,A -85,B 0,C 180,E1 -1386.763,E2 -1386.763} C_VEL
LIN {X 0,Y 587.121,Z 648.987,A -85,B 0,C 180,E1 -1387.81,E2 -1387.81} C_VEL
LIN {X 0,Y 587.111,Z 650.354,A -85,B 0,C 180,E1 -1389.378,E2 -1389.378} C_VEL
LIN {X 0,Y 587.139,Z 650.455,A -85,B 0,C 180,E1 -1390.269,E2 -1390.269} C_VEL
LIN {X 0,Y 587.122,Z 650.077,A -85,B 0,C 180,E1 -1391.176,E2 -1391.176} C_VEL
LIN {X 0,Y 587.168,Z 649.209,A -85,B 0,C 180,E1 -1392.089,E2 -1392.089} C_VEL
LIN {X 0,Y 587.148,Z 647.67,A -85,B 0,C 180,E1 -1393.1,E2 -1393.1} C_VEL
LIN {X 0,Y 587.166,Z 644.459,A -85,B 0,C 180,E1 -1394.485,E2 -1394.485} C_VEL
LIN {X 0,Y 587.185,Z 639.379,A -85,B 0,C 180,E1 -1396.036,E2 -1396.036} C_VEL
LIN {X 0,Y 587.219,Z 633.213,A -85,B 0,C 180,E1 -1397.452,E2 -1397.452} C_VEL
LIN {X 0,Y 587.232,Z 625.656,A -85,B 0,C 180,E1 -1398.834,E2 -1398.834} C_VEL
LIN {X 0,Y 587.309,Z 616.857,A -85,B 0,C 180,E1 -1400.145,E2 -1400.145} C_VEL
LIN {X 0,Y 587.416,Z 606.575,A -85,B 0,C 180,E1 -1401.41,E2 -1401.41} C_VEL
LIN {X 0,Y 587.489,Z 595.864,A -85,B 0,C 180,E1 -1402.511,E2 -1402.511} C_VEL
LIN {X 0,Y 587.616,Z 584.598,A -85,B 0,C 180,E1 -1403.486,E2 -1403.486} C_VEL
LIN {X 0,Y 587.748,Z 571.972,A -85,B 0,C 180,E1 -1404.401,E2 -1404.401} C_VEL
LIN {X 0,Y 587.855,Z 558.078,A -85,B 0,C 180,E1 -1405.231,E2 -1405.231} C_VEL
LIN {X 0,Y 588.029,Z 543.486,A -85,B 0,C 180,E1 -1405.927,E2 -1405.927} C_VEL
LIN {X 0,Y 588.161,Z 529.389,A -85,B 0,C 180,E1 -1406.451,E2 -1406.451} C_VEL
LIN {X 0,Y 588.228,Z 513.922,A -85,B 0,C 180,E1 -1406.876,E2 -1406.876} C_VEL
LIN {X 0,Y 588.289,Z 498.265,A -85,B 0,C 180,E1 -1407.154,E2 -1407.154} C_VEL
LIN {X 0,Y 588.509,Z 344.882,A -85,B 0,C 180,E1 -1409.077,E2 -1409.077} C_VEL
LIN {X 0,Y 587.572,Z 340.49,A -85,B 0,C 180,E1 -1409.167,E2 -1409.167} C_VEL
LIN {X 0,Y 587.641,Z 329.216,A -85,B 0,C 180,E1 -1410.816,E2 -1410.816} C_VEL
LIN {X 0,Y 587.278,Z 326.957,A -85,B 0,C 180,E1 -1411.174,E2 -1411.174} C_VEL
LIN {X 0,Y 587.294,Z 326.958,A -85,B 0,C 180,E1 -1413.833,E2 -1413.833} C_VEL
LIN {X 0,Y 587.297,Z 326.949,A -85,B 0,C 180,E1 -1416.74,E2 -1416.74} C_VEL
LIN {X 0,Y 587.307,Z 326.955,A -85,B 0,C 180,E1 -1419.694,E2 -1419.694} C_VEL
LIN {X 0,Y 587.281,Z 326.959,A -85,B 0,C 180,E1 -1421.872,E2 -1421.872} C_VEL
LIN {X 0,Y 587.302,Z 326.948,A -85,B 0,C 180,E1 -1424.736,E2 -1424.736} C_VEL
LIN {X 0,Y 587.293,Z 326.949,A -85,B 0,C 180,E1 -1426.857,E2 -1426.857} C_VEL
LIN {X 0,Y 587.33,Z 326.954,A -85,B 0,C 180,E1 -1429.66,E2 -1429.66} C_VEL
LIN {X 0,Y 587.313,Z 326.946,A -85,B 0,C 180,E1 -1432.436,E2 -1432.436} C_VEL
LIN {X 0,Y 587.345,Z 326.946,A -85,B 0,C 180,E1 -1435.195,E2 -1435.195} C_VEL
LIN {X 0,Y 587.372,Z 326.943,A -85,B 0,C 180,E1 -1437.943,E2 -1437.943} C_VEL
LIN {X 0,Y 587.369,Z 326.939,A -85,B 0,C 180,E1 -1440.685,E2 -1440.685} C_VEL
LIN {X 0,Y 587.326,Z 326.954,A -85,B 0,C 180,E1 -1443.43,E2 -1443.43} C_VEL
LIN {X 0,Y 587.315,Z 326.947,A -85,B 0,C 180,E1 -1446.182,E2 -1446.182} C_VEL
LIN {X 0,Y 587.342,Z 326.943,A -85,B 0,C 180,E1 -1448.255,E2 -1448.255} C_VEL
LIN {X 0,Y 587.352,Z 326.947,A -85,B 0,C 180,E1 -1451.133,E2 -1451.133} C_VEL
LIN {X 0,Y 587.343,Z 326.942,A -85,B 0,C 180,E1 -1454.251,E2 -1454.251} C_VEL
LIN {X 0,Y 587.347,Z 326.95,A -85,B 0,C 180,E1 -1457.406,E2 -1457.406} C_VEL
LIN {X 0,Y 587.323,Z 326.945,A -85,B 0,C 180,E1 -1460.305,E2 -1460.305} C_VEL
LIN {X 0,Y 587.316,Z 326.955,A -85,B 0,C 180,E1 -1463.259,E2 -1463.259} C_VEL
LIN {X 0,Y 587.332,Z 326.948,A -85,B 0,C 180,E1 -1465.517,E2 -1465.517} C_VEL
LIN {X 0,Y 587.347,Z 326.943,A -85,B 0,C 180,E1 -1467.818,E2 -1467.818} C_VEL
LIN {X 0,Y 587.338,Z 326.944,A -85,B 0,C 180,E1 -1470.51,E2 -1470.51} C_VEL
LIN {X 0,Y 587.334,Z 326.948,A -85,B 0,C 180,E1 -1473.397,E2 -1473.397} C_VEL
LIN {X 0,Y 587.293,Z 326.949,A -85,B 0,C 180,E1 -1475.9,E2 -1475.9} C_VEL
LIN {X 0,Y 587.332,Z 326.946,A -85,B 0,C 180,E1 -1478.479,E2 -1478.479} C_VEL
LIN {X 0,Y 587.338,Z 326.95,A -85,B 0,C 180,E1 -1481.157,E2 -1481.157} C_VEL
LIN {X 0,Y 587.328,Z 326.945,A -85,B 0,C 180,E1 -1484.113,E2 -1484.113} C_VEL
LIN {X 0,Y 587.321,Z 326.954,A -85,B 0,C 180,E1 -1486.994,E2 -1486.994} C_VEL
LIN {X 0,Y 587.318,Z 326.946,A -85,B 0,C 180,E1 -1489.746,E2 -1489.746} C_VEL
LIN {X 0,Y 587.346,Z 326.946,A -85,B 0,C 180,E1 -1492.392,E2 -1492.392} C_VEL
LIN {X 0,Y 587.358,Z 326.941,A -85,B 0,C 180,E1 -1495.779,E2 -1495.779} C_VEL
LIN {X 0,Y 587.339,Z 326.946,A -85,B 0,C 180,E1 -1498.231,E2 -1498.231} C_VEL
LIN {X 0,Y 587.346,Z 326.952,A -85,B 0,C 180,E1 -1500.867,E2 -1500.867} C_VEL
LIN {X 0,Y 587.393,Z 327.114,A -85,B 0,C 180,E1 -1502.861,E2 -1502.861} C_VEL
LIN {X 0,Y 588.475,Z 333.062,A -85,B 0,C 180,E1 -1503.599,E2 -1503.599} C_VEL
LIN {X 0,Y 588.231,Z 357.93,A -85,B 0,C 180,E1 -1506.406,E2 -1506.406} C_VEL
LIN {X 0,Y 587.967,Z 384.588,A -85,B 0,C 180,E1 -1509.352,E2 -1509.352} C_VEL
LIN {X 0,Y 587.825,Z 398.434,A -85,B 0,C 180,E1 -1510.861,E2 -1510.861} C_VEL
LIN {X 0,Y 588.62,Z 402.939,A -85,B 0,C 180,E1 -1510.947,E2 -1510.947} C_VEL
LIN {X 0,Y 588.298,Z 565.405,A -85,B 0,C 180,E1 -1513,E2 -1513} C_VEL
LIN {X 0,Y 588.21,Z 581.474,A -85,B 0,C 180,E1 -1513.358,E2 -1513.358} C_VEL
LIN {X 0,Y 588.072,Z 596.037,A -85,B 0,C 180,E1 -1513.823,E2 -1513.823} C_VEL
LIN {X 0,Y 587.989,Z 609.758,A -85,B 0,C 180,E1 -1514.399,E2 -1514.399} C_VEL
LIN {X 0,Y 587.829,Z 623.233,A -85,B 0,C 180,E1 -1515.105,E2 -1515.105} C_VEL
LIN {X 0,Y 587.741,Z 636.109,A -85,B 0,C 180,E1 -1515.929,E2 -1515.929} C_VEL
LIN {X 0,Y 587.582,Z 648.283,A -85,B 0,C 180,E1 -1516.864,E2 -1516.864} C_VEL
LIN {X 0,Y 587.455,Z 659.745,A -85,B 0,C 180,E1 -1517.915,E2 -1517.915} C_VEL
LIN {X 0,Y 587.348,Z 669.387,A -85,B 0,C 180,E1 -1518.962,E2 -1518.962} C_VEL
LIN {X 0,Y 587.305,Z 678.854,A -85,B 0,C 180,E1 -1520.181,E2 -1520.181} C_VEL
LIN {X 0,Y 587.264,Z 686.73,A -85,B 0,C 180,E1 -1521.396,E2 -1521.396} C_VEL
LIN {X 0,Y 587.215,Z 694.087,A -85,B 0,C 180,E1 -1522.78,E2 -1522.78} C_VEL
LIN {X 0,Y 587.226,Z 699.923,A -85,B 0,C 180,E1 -1524.161,E2 -1524.161} C_VEL
LIN {X 0,Y 587.136,Z 703.383,A -85,B 0,C 180,E1 -1525.193,E2 -1525.193} C_VEL
LIN {X 0,Y 587.18,Z 706.887,A -85,B 0,C 180,E1 -1526.569,E2 -1526.569} C_VEL
LIN {X 0,Y 587.139,Z 709.193,A -85,B 0,C 180,E1 -1527.942,E2 -1527.942} C_VEL
LIN {X 0,Y 587.135,Z 710.35,A -85,B 0,C 180,E1 -1529.314,E2 -1529.314} C_VEL
LIN {X 0,Y 587.135,Z 710.35,A -85,B 0,C 180,E1 -1530.686,E2 -1530.686} C_VEL
LIN {X 0,Y 587.139,Z 709.193,A -85,B 0,C 180,E1 -1532.058,E2 -1532.058} C_VEL
LIN {X 0,Y 587.18,Z 706.887,A -85,B 0,C 180,E1 -1533.431,E2 -1533.431} C_VEL
LIN {X 0,Y 587.136,Z 703.385,A -85,B 0,C 180,E1 -1534.806,E2 -1534.806} C_VEL
LIN {X 0,Y 587.179,Z 698.609,A -85,B 0,C 180,E1 -1536.184,E2 -1536.184} C_VEL
LIN {X 0,Y 587.23,Z 692.426,A -85,B 0,C 180,E1 -1537.565,E2 -1537.565} C_VEL
LIN {X 0,Y 587.265,Z 684.653,A -85,B 0,C 180,E1 -1538.95,E2 -1538.95} C_VEL
LIN {X 0,Y 587.352,Z 676.372,A -85,B 0,C 180,E1 -1540.165,E2 -1540.165} C_VEL
LIN {X 0,Y 587.399,Z 666.398,A -85,B 0,C 180,E1 -1541.385,E2 -1541.385} C_VEL
LIN {X 0,Y 587.522,Z 656.194,A -85,B 0,C 180,E1 -1542.434,E2 -1542.434} C_VEL
LIN {X 0,Y 587.629,Z 644.022,A -85,B 0,C 180,E1 -1543.486,E2 -1543.486} C_VEL
LIN {X 0,Y 587.773,Z 631.061,A -85,B 0,C 180,E1 -1544.416,E2 -1544.416} C_VEL
LIN {X 0,Y 587.887,Z 616.872,A -85,B 0,C 180,E1 -1545.248,E2 -1545.248} C_VEL
LIN {X 0,Y 588.049,Z 602.804,A -85,B 0,C 180,E1 -1545.91,E2 -1545.91} C_VEL
LIN {X 0,Y 588.171,Z 588.313,A -85,B 0,C 180,E1 -1546.441,E2 -1546.441} C_VEL
LIN {X 0,Y 588.274,Z 573.307,A -85,B 0,C 180,E1 -1546.844,E2 -1546.844} C_VEL
LIN {X 0,Y 588.319,Z 558.133,A -85,B 0,C 180,E1 -1547.109,E2 -1547.109} C_VEL
LIN {X 0,Y 588.526,Z 401.911,A -85,B 0,C 180,E1 -1549.069,E2 -1549.069} C_VEL
LIN {X 0,Y 587.835,Z 398.332,A -85,B 0,C 180,E1 -1549.15,E2 -1549.15} C_VEL
LIN {X 0,Y 588.022,Z 374.597,A -85,B 0,C 180,E1 -1551.747,E2 -1551.747} C_VEL
LIN {X 0,Y 588.289,Z 349.606,A -85,B 0,C 180,E1 -1554.528,E2 -1554.528} C_VEL
LIN {X 0,Y 588.471,Z 333.071,A -85,B 0,C 180,E1 -1556.4,E2 -1556.4} C_VEL
LIN {X 0,Y 587.953,Z 329.537,A -85,B 0,C 180,E1 -1556.832,E2 -1556.832} C_VEL
LIN {X 0,Y 587.367,Z 326.945,A -85,B 0,C 180,E1 -1557.187,E2 -1557.187} C_VEL
LIN {X 0,Y 587.331,Z 326.945,A -85,B 0,C 180,E1 -1560.17,E2 -1560.17} C_VEL
LIN {X 0,Y 587.332,Z 326.945,A -85,B 0,C 180,E1 -1562.579,E2 -1562.579} C_VEL
LIN {X 0,Y 587.32,Z 326.952,A -85,B 0,C 180,E1 -1565.056,E2 -1565.056} C_VEL
LIN {X 0,Y 587.338,Z 326.946,A -85,B 0,C 180,E1 -1567.838,E2 -1567.838} C_VEL
LIN {X 0,Y 587.314,Z 326.945,A -85,B 0,C 180,E1 -1570.254,E2 -1570.254} C_VEL
LIN {X 0,Y 587.317,Z 326.952,A -85,B 0,C 180,E1 -1573.006,E2 -1573.006} C_VEL
LIN {X 0,Y 587.324,Z 326.945,A -85,B 0,C 180,E1 -1575.886,E2 -1575.886} C_VEL
LIN {X 0,Y 587.335,Z 326.947,A -85,B 0,C 180,E1 -1578.843,E2 -1578.843} C_VEL
LIN {X 0,Y 587.328,Z 326.949,A -85,B 0,C 180,E1 -1581.521,E2 -1581.521} C_VEL
LIN {X 0,Y 587.349,Z 326.942,A -85,B 0,C 180,E1 -1584.455,E2 -1584.455} C_VEL
LIN {X 0,Y 587.335,Z 326.949,A -85,B 0,C 180,E1 -1586.888,E2 -1586.888} C_VEL
LIN {X 0,Y 587.331,Z 326.944,A -85,B 0,C 180,E1 -1589.83,E2 -1589.83} C_VEL
LIN {X 0,Y 587.348,Z 326.942,A -85,B 0,C 180,E1 -1592.307,E2 -1592.307} C_VEL
LIN {X 0,Y 587.348,Z 326.949,A -85,B 0,C 180,E1 -1595.242,E2 -1595.242} C_VEL
LIN {X 0,Y 587.319,Z 326.945,A -85,B 0,C 180,E1 -1598.226,E2 -1598.226} C_VEL
LIN {X 0,Y 587.346,Z 326.95,A -85,B 0,C 180,E1 -1601.151,E2 -1601.151} C_VEL
LIN {X 0,Y 587.322,Z 326.944,A -85,B 0,C 180,E1 -1604.025,E2 -1604.025} C_VEL
LIN {X 0,Y 587.358,Z 326.94,A -85,B 0,C 180,E1 -1606.154,E2 -1606.154} C_VEL
LIN {X 0,Y 587.339,Z 326.953,A -85,B 0,C 180,E1 -1608.963,E2 -1608.963} C_VEL
LIN {X 0,Y 587.363,Z 326.94,A -85,B 0,C 180,E1 -1611.745,E2 -1611.745} C_VEL
LIN {X 0,Y 587.362,Z 326.943,A -85,B 0,C 180,E1 -1614.507,E2 -1614.507} C_VEL
LIN {X 0,Y 587.367,Z 326.944,A -85,B 0,C 180,E1 -1617.257,E2 -1617.257} C_VEL
LIN {X 0,Y 587.382,Z 326.937,A -85,B 0,C 180,E1 -1620,E2 -1620} C_VEL
LIN {X 0,Y 587.37,Z 326.947,A -85,B 0,C 180,E1 -1622.744,E2 -1622.744} C_VEL
LIN {X 0,Y 587.357,Z 326.942,A -85,B 0,C 180,E1 -1625.493,E2 -1625.493} C_VEL
LIN {X 0,Y 587.368,Z 326.941,A -85,B 0,C 180,E1 -1628.255,E2 -1628.255} C_VEL
LIN {X 0,Y 587.346,Z 326.947,A -85,B 0,C 180,E1 -1631.134,E2 -1631.134} C_VEL
LIN {X 0,Y 587.364,Z 326.942,A -85,B 0,C 180,E1 -1634.261,E2 -1634.261} C_VEL
LIN {X 0,Y 587.347,Z 326.943,A -85,B 0,C 180,E1 -1637.406,E2 -1637.406} C_VEL
LIN {X 0,Y 587.309,Z 326.948,A -85,B 0,C 180,E1 -1638.313,E2 -1638.313} C_VEL
LIN {X 0,Y 586.666,Z 327.035,A -85,B 0,C 180,E1 -1638.885,E2 -1638.885} C_VEL
LIN {X 0,Y 583.841,Z 327.387,A -85,B 0,C 180,E1 -1639.814,E2 -1639.814} C_VEL
LIN {X 0,Y 581.43,Z 327.686,A -85,B 0,C 180,E1 -1640.561,E2 -1640.561} C_VEL
LIN {X 0,Y 580.376,Z 327.814,A -85,B 0,C 180,E1 -1641.137,E2 -1641.137} C_VEL
LIN {X 0,Y 580.281,Z 327.823,A -85,B 0,C 180,E1 -1641.332,E2 -1641.332} C_VEL
LIN {X 0,Y 580.297,Z 327.823,A -85,B 0,C 180,E1 -1644.317,E2 -1644.317} C_VEL
LIN {X 0,Y 580.271,Z 327.832,A -85,B 0,C 180,E1 -1646.624,E2 -1646.624} C_VEL
LIN {X 0,Y 580.3,Z 327.821,A -85,B 0,C 180,E1 -1649.31,E2 -1649.31} C_VEL
LIN {X 0,Y 580.297,Z 327.823,A -85,B 0,C 180,E1 -1652.201,E2 -1652.201} C_VEL
LIN {X 0,Y 580.288,Z 327.831,A -85,B 0,C 180,E1 -1654.697,E2 -1654.697} C_VEL
LIN {X 0,Y 580.298,Z 327.821,A -85,B 0,C 180,E1 -1657.269,E2 -1657.269} C_VEL
LIN {X 0,Y 580.29,Z 327.825,A -85,B 0,C 180,E1 -1660.271,E2 -1660.271} C_VEL
LIN {X 0,Y 580.272,Z 327.831,A -85,B 0,C 180,E1 -1662.707,E2 -1662.707} C_VEL
LIN {X 0,Y 580.258,Z 327.824,A -85,B 0,C 180,E1 -1665.611,E2 -1665.611} C_VEL
LIN {X 0,Y 580.275,Z 327.827,A -85,B 0,C 180,E1 -1668.231,E2 -1668.231} C_VEL
LIN {X 0,Y 580.27,Z 327.827,A -85,B 0,C 180,E1 -1670.965,E2 -1670.965} C_VEL
LIN {X 0,Y 580.248,Z 327.826,A -85,B 0,C 180,E1 -1673.595,E2 -1673.595} C_VEL
LIN {X 0,Y 580.313,Z 327.822,A -85,B 0,C 180,E1 -1676.146,E2 -1676.146} C_VEL
LIN {X 0,Y 580.269,Z 327.831,A -85,B 0,C 180,E1 -1678.615,E2 -1678.615} C_VEL
LIN {X 0,Y 580.286,Z 327.823,A -85,B 0,C 180,E1 -1681.024,E2 -1681.024} C_VEL
LIN {X 0,Y 580.266,Z 327.829,A -85,B 0,C 180,E1 -1684.15,E2 -1684.15} C_VEL
LIN {X 0,Y 580.259,Z 327.826,A -85,B 0,C 180,E1 -1687,E2 -1687} C_VEL
LIN {X 0,Y 580.265,Z 327.824,A -85,B 0,C 180,E1 -1689.437,E2 -1689.437} C_VEL
LIN {X 0,Y 580.246,Z 327.827,A -85,B 0,C 180,E1 -1691.645,E2 -1691.645} C_VEL
LIN {X 0,Y 580.275,Z 327.83,A -85,B 0,C 180,E1 -1694.547,E2 -1694.547} C_VEL
LIN {X 0,Y 580.246,Z 327.831,A -85,B 0,C 180,E1 -1696.696,E2 -1696.696} C_VEL
LIN {X 0,Y 580.31,Z 327.821,A -85,B 0,C 180,E1 -1698.827,E2 -1698.827} C_VEL
LIN {X 0,Y 580.306,Z 327.82,A -85,B 0,C 180,E1 -1701.644,E2 -1701.644} C_VEL
LIN {X 0,Y 580.306,Z 327.827,A -85,B 0,C 180,E1 -1704.44,E2 -1704.44} C_VEL
LIN {X 0,Y 580.34,Z 327.819,A -85,B 0,C 180,E1 -1707.918,E2 -1707.918} C_VEL
LIN {X 0,Y 580.343,Z 327.817,A -85,B 0,C 180,E1 -1710.694,E2 -1710.694} C_VEL
LIN {X 0,Y 580.312,Z 327.82,A -85,B 0,C 180,E1 -1712.777,E2 -1712.777} C_VEL
LIN {X 0,Y 580.296,Z 327.821,A -85,B 0,C 180,E1 -1715.56,E2 -1715.56} C_VEL
LIN {X 0,Y 580.302,Z 327.827,A -85,B 0,C 180,E1 -1718.357,E2 -1718.357} C_VEL
LIN {X 0,Y 580.272,Z 327.823,A -85,B 0,C 180,E1 -1721.174,E2 -1721.174} C_VEL
LIN {X 0,Y 580.31,Z 327.827,A -85,B 0,C 180,E1 -1724.018,E2 -1724.018} C_VEL
LIN {X 0,Y 580.236,Z 327.83,A -85,B 0,C 180,E1 -1726.9,E2 -1726.9} C_VEL
LIN {X 0,Y 580.283,Z 327.973,A -85,B 0,C 180,E1 -1728.812,E2 -1728.812} C_VEL
LIN {X 0,Y 580.744,Z 333.187,A -85,B 0,C 180,E1 -1729.607,E2 -1729.607} C_VEL
LIN {X 0,Y 580.639,Z 340.467,A -85,B 0,C 180,E1 -1730.682,E2 -1730.682} C_VEL
LIN {X 0,Y 581.871,Z 346.818,A -85,B 0,C 180,E1 -1730.812,E2 -1730.812} C_VEL
LIN {X 0,Y 581.482,Z 505.564,A -85,B 0,C 180,E1 -1732.842,E2 -1732.842} C_VEL
LIN {X 0,Y 581.435,Z 521.303,A -85,B 0,C 180,E1 -1733.198,E2 -1733.198} C_VEL
LIN {X 0,Y 581.254,Z 536.887,A -85,B 0,C 180,E1 -1733.705,E2 -1733.705} C_VEL
LIN {X 0,Y 581.117,Z 550.293,A -85,B 0,C 180,E1 -1734.28,E2 -1734.28} C_VEL
LIN {X 0,Y 580.886,Z 564.714,A -85,B 0,C 180,E1 -1735.053,E2 -1735.053} C_VEL
LIN {X 0,Y 580.757,Z 577.652,A -85,B 0,C 180,E1 -1735.91,E2 -1735.91} C_VEL
LIN {X 0,Y 580.601,Z 590.068,A -85,B 0,C 180,E1 -1736.899,E2 -1736.899} C_VEL
LIN {X 0,Y 580.441,Z 601.576,A -85,B 0,C 180,E1 -1737.996,E2 -1737.996} C_VEL
LIN {X 0,Y 580.334,Z 611.665,A -85,B 0,C 180,E1 -1739.144,E2 -1739.144} C_VEL
LIN {X 0,Y 580.231,Z 620.752,A -85,B 0,C 180,E1 -1740.378,E2 -1740.378} C_VEL
LIN {X 0,Y 580.192,Z 628.81,A -85,B 0,C 180,E1 -1741.698,E2 -1741.698} C_VEL
LIN {X 0,Y 580.1,Z 635.476,A -85,B 0,C 180,E1 -1743.037,E2 -1743.037} C_VEL
LIN {X 0,Y 580.085,Z 640.15,A -85,B 0,C 180,E1 -1744.197,E2 -1744.197} C_VEL
LIN {X 0,Y 580.064,Z 644.484,A -85,B 0,C 180,E1 -1745.561,E2 -1745.561} C_VEL
LIN {X 0,Y 580.035,Z 647.56,A -85,B 0,C 180,E1 -1746.899,E2 -1746.899} C_VEL
LIN {X 0,Y 580.017,Z 649.424,A -85,B 0,C 180,E1 -1748.168,E2 -1748.168} C_VEL
LIN {X 0,Y 580.018,Z 650.246,A -85,B 0,C 180,E1 -1749.151,E2 -1749.151} C_VEL
LIN {X 0,Y 580.038,Z 650.462,A -85,B 0,C 180,E1 -1750.24,E2 -1750.24} C_VEL
LIN {X 0,Y 580.053,Z 649.575,A -85,B 0,C 180,E1 -1751.789,E2 -1751.789} C_VEL
LIN {X 0,Y 580.059,Z 648.34,A -85,B 0,C 180,E1 -1752.727,E2 -1752.727} C_VEL
LIN {X 0,Y 580.032,Z 646.55,A -85,B 0,C 180,E1 -1753.681,E2 -1753.681} C_VEL
LIN {X 0,Y 580.093,Z 643.113,A -85,B 0,C 180,E1 -1754.999,E2 -1754.999} C_VEL
LIN {X 0,Y 580.103,Z 638.525,A -85,B 0,C 180,E1 -1756.325,E2 -1756.325} C_VEL
LIN {X 0,Y 580.134,Z 632.72,A -85,B 0,C 180,E1 -1757.645,E2 -1757.645} C_VEL
LIN {X 0,Y 580.182,Z 625.808,A -85,B 0,C 180,E1 -1758.915,E2 -1758.915} C_VEL
LIN {X 0,Y 580.268,Z 616.882,A -85,B 0,C 180,E1 -1760.265,E2 -1760.265} C_VEL
LIN {X 0,Y 580.393,Z 607.692,A -85,B 0,C 180,E1 -1761.419,E2 -1761.419} C_VEL
LIN {X 0,Y 580.475,Z 597.263,A -85,B 0,C 180,E1 -1762.526,E2 -1762.526} C_VEL
LIN {X 0,Y 580.664,Z 584.895,A -85,B 0,C 180,E1 -1763.625,E2 -1763.625} C_VEL
LIN {X 0,Y 580.807,Z 571.661,A -85,B 0,C 180,E1 -1764.598,E2 -1764.598} C_VEL
LIN {X 0,Y 580.99,Z 557.806,A -85,B 0,C 180,E1 -1765.429,E2 -1765.429} C_VEL
LIN {X 0,Y 581.184,Z 543.978,A -85,B 0,C 180,E1 -1766.098,E2 -1766.098} C_VEL
LIN {X 0,Y 581.329,Z 529.778,A -85,B 0,C 180,E1 -1766.636,E2 -1766.636} C_VEL
LIN {X 0,Y 581.423,Z 514.639,A -85,B 0,C 180,E1 -1767.061,E2 -1767.061} C_VEL
LIN {X 0,Y 581.523,Z 498.842,A -85,B 0,C 180,E1 -1767.351,E2 -1767.351} C_VEL
LIN {X 0,Y 581.806,Z 346,A -85,B 0,C 180,E1 -1769.29,E2 -1769.29} C_VEL
LIN {X 0,Y 580.642,Z 340.411,A -85,B 0,C 180,E1 -1769.416,E2 -1769.416} C_VEL
LIN {X 0,Y 580.72,Z 330.869,A -85,B 0,C 180,E1 -1770.829,E2 -1770.829} C_VEL
LIN {X 0,Y 580.247,Z 327.834,A -85,B 0,C 180,E1 -1771.318,E2 -1771.318} C_VEL
LIN {X 0,Y 580.239,Z 327.835,A -85,B 0,C 180,E1 -1774.148,E2 -1774.148} C_VEL
LIN {X 0,Y 580.244,Z 327.828,A -85,B 0,C 180,E1 -1777.003,E2 -1777.003} C_VEL
LIN {X 0,Y 580.249,Z 327.83,A -85,B 0,C 180,E1 -1779.436,E2 -1779.436} C_VEL
LIN {X 0,Y 580.241,Z 327.835,A -85,B 0,C 180,E1 -1781.644,E2 -1781.644} C_VEL
LIN {X 0,Y 580.27,Z 327.824,A -85,B 0,C 180,E1 -1784.546,E2 -1784.546} C_VEL
LIN {X 0,Y 580.253,Z 327.826,A -85,B 0,C 180,E1 -1786.695,E2 -1786.695} C_VEL
LIN {X 0,Y 580.309,Z 327.819,A -85,B 0,C 180,E1 -1788.827,E2 -1788.827} C_VEL
LIN {X 0,Y 580.306,Z 327.829,A -85,B 0,C 180,E1 -1791.643,E2 -1791.643} C_VEL
LIN {X 0,Y 580.301,Z 327.82,A -85,B 0,C 180,E1 -1794.44,E2 -1794.44} C_VEL
LIN {X 0,Y 580.324,Z 327.821,A -85,B 0,C 180,E1 -1797.223,E2 -1797.223} C_VEL
LIN {X 0,Y 580.353,Z 327.816,A -85,B 0,C 180,E1 -1800,E2 -1800} C_VEL
LIN {X 0,Y 580.322,Z 327.818,A -85,B 0,C 180,E1 -1802.776,E2 -1802.776} C_VEL
LIN {X 0,Y 580.318,Z 327.826,A -85,B 0,C 180,E1 -1805.56,E2 -1805.56} C_VEL
LIN {X 0,Y 580.31,Z 327.819,A -85,B 0,C 180,E1 -1808.356,E2 -1808.356} C_VEL
LIN {X 0,Y 580.304,Z 327.826,A -85,B 0,C 180,E1 -1811.191,E2 -1811.191} C_VEL
LIN {X 0,Y 580.318,Z 327.819,A -85,B 0,C 180,E1 -1814.017,E2 -1814.017} C_VEL
LIN {X 0,Y 580.315,Z 327.821,A -85,B 0,C 180,E1 -1816.913,E2 -1816.913} C_VEL
LIN {X 0,Y 580.287,Z 327.823,A -85,B 0,C 180,E1 -1819.823,E2 -1819.823} C_VEL
LIN {X 0,Y 580.27,Z 327.824,A -85,B 0,C 180,E1 -1822.053,E2 -1822.053} C_VEL
LIN {X 0,Y 580.307,Z 327.827,A -85,B 0,C 180,E1 -1825.08,E2 -1825.08} C_VEL
LIN {X 0,Y 580.298,Z 327.82,A -85,B 0,C 180,E1 -1828.185,E2 -1828.185} C_VEL
LIN {X 0,Y 580.286,Z 327.825,A -85,B 0,C 180,E1 -1830.694,E2 -1830.694} C_VEL
LIN {X 0,Y 580.303,Z 327.826,A -85,B 0,C 180,E1 -1833.316,E2 -1833.316} C_VEL
LIN {X 0,Y 580.247,Z 327.827,A -85,B 0,C 180,E1 -1835.756,E2 -1835.756} C_VEL
LIN {X 0,Y 580.29,Z 327.821,A -85,B 0,C 180,E1 -1838.146,E2 -1838.146} C_VEL
LIN {X 0,Y 580.3,Z 327.828,A -85,B 0,C 180,E1 -1840.843,E2 -1840.843} C_VEL
LIN {X 0,Y 580.28,Z 327.823,A -85,B 0,C 180,E1 -1843.658,E2 -1843.658} C_VEL
LIN {X 0,Y 580.286,Z 327.827,A -85,B 0,C 180,E1 -1846.608,E2 -1846.608} C_VEL
LIN {X 0,Y 580.3,Z 327.826,A -85,B 0,C 180,E1 -1849.156,E2 -1849.156} C_VEL
LIN {X 0,Y 580.29,Z 327.822,A -85,B 0,C 180,E1 -1851.927,E2 -1851.927} C_VEL
LIN {X 0,Y 580.251,Z 327.831,A -85,B 0,C 180,E1 -1854.452,E2 -1854.452} C_VEL
LIN {X 0,Y 580.29,Z 327.828,A -85,B 0,C 180,E1 -1856.975,E2 -1856.975} C_VEL
LIN {X 0,Y 580.296,Z 327.823,A -85,B 0,C 180,E1 -1859.425,E2 -1859.425} C_VEL
LIN {X 0,Y 580.29,Z 327.828,A -85,B 0,C 180,E1 -1862.143,E2 -1862.143} C_VEL
LIN {X 0,Y 580.337,Z 327.937,A -85,B 0,C 180,E1 -1862.614,E2 -1862.614} C_VEL
LIN {X 0,Y 581.696,Z 334.605,A -85,B 0,C 180,E1 -1863.446,E2 -1863.446} C_VEL
LIN {X 0,Y 581.438,Z 357.93,A -85,B 0,C 180,E1 -1866.113,E2 -1866.113} C_VEL
LIN {X 0,Y 581.109,Z 384.588,A -85,B 0,C 180,E1 -1869.097,E2 -1869.097} C_VEL
LIN {X 0,Y 580.942,Z 398.414,A -85,B 0,C 180,E1 -1870.623,E2 -1870.623} C_VEL
LIN {X 0,Y 581.91,Z 404.735,A -85,B 0,C 180,E1 -1870.742,E2 -1870.742} C_VEL
LIN {X 0,Y 581.534,Z 564.72,A -85,B 0,C 180,E1 -1872.784,E2 -1872.784} C_VEL
LIN {X 0,Y 581.416,Z 580.697,A -85,B 0,C 180,E1 -1873.135,E2 -1873.135} C_VEL
LIN {X 0,Y 581.242,Z 596.035,A -85,B 0,C 180,E1 -1873.627,E2 -1873.627} C_VEL
LIN {X 0,Y 581.125,Z 609.761,A -85,B 0,C 180,E1 -1874.21,E2 -1874.21} C_VEL
LIN {X 0,Y 580.944,Z 623.235,A -85,B 0,C 180,E1 -1874.924,E2 -1874.924} C_VEL
LIN {X 0,Y 580.805,Z 636.475,A -85,B 0,C 180,E1 -1875.783,E2 -1875.783} C_VEL
LIN {X 0,Y 580.608,Z 648.285,A -85,B 0,C 180,E1 -1876.703,E2 -1876.703} C_VEL
LIN {X 0,Y 580.479,Z 659.746,A -85,B 0,C 180,E1 -1877.767,E2 -1877.767} C_VEL
LIN {X 0,Y 580.307,Z 670.454,A -85,B 0,C 180,E1 -1878.953,E2 -1878.953} C_VEL
LIN {X 0,Y 580.269,Z 678.855,A -85,B 0,C 180,E1 -1880.061,E2 -1880.061} C_VEL
LIN {X 0,Y 580.213,Z 686.731,A -85,B 0,C 180,E1 -1881.291,E2 -1881.291} C_VEL
LIN {X 0,Y 580.131,Z 694.087,A -85,B 0,C 180,E1 -1882.692,E2 -1882.692} C_VEL
LIN {X 0,Y 580.131,Z 699.922,A -85,B 0,C 180,E1 -1884.089,E2 -1884.089} C_VEL
LIN {X 0,Y 580.041,Z 703.384,A -85,B 0,C 180,E1 -1885.134,E2 -1885.134} C_VEL
LIN {X 0,Y 580.105,Z 706.888,A -85,B 0,C 180,E1 -1886.527,E2 -1886.527} C_VEL
LIN {X 0,Y 580.038,Z 709.192,A -85,B 0,C 180,E1 -1887.917,E2 -1887.917} C_VEL
LIN {X 0,Y 580.036,Z 710.349,A -85,B 0,C 180,E1 -1889.305,E2 -1889.305} C_VEL
LIN {X 0,Y 580.036,Z 710.349,A -85,B 0,C 180,E1 -1890.694,E2 -1890.694} C_VEL
LIN {X 0,Y 580.038,Z 709.192,A -85,B 0,C 180,E1 -1892.083,E2 -1892.083} C_VEL
LIN {X 0,Y 580.105,Z 706.887,A -85,B 0,C 180,E1 -1893.473,E2 -1893.473} C_VEL
LIN {X 0,Y 580.041,Z 703.386,A -85,B 0,C 180,E1 -1894.865,E2 -1894.865} C_VEL
LIN {X 0,Y 580.092,Z 698.609,A -85,B 0,C 180,E1 -1896.26,E2 -1896.26} C_VEL
LIN {X 0,Y 580.165,Z 692.425,A -85,B 0,C 180,E1 -1897.657,E2 -1897.657} C_VEL
LIN {X 0,Y 580.206,Z 684.652,A -85,B 0,C 180,E1 -1899.06,E2 -1899.06} C_VEL
LIN {X 0,Y 580.309,Z 676.372,A -85,B 0,C 180,E1 -1900.29,E2 -1900.29} C_VEL
LIN {X 0,Y 580.382,Z 666.398,A -85,B 0,C 180,E1 -1901.525,E2 -1901.525} C_VEL
LIN {X 0,Y 580.541,Z 656.193,A -85,B 0,C 180,E1 -1902.586,E2 -1902.586} C_VEL
LIN {X 0,Y 580.677,Z 644.023,A -85,B 0,C 180,E1 -1903.651,E2 -1903.651} C_VEL
LIN {X 0,Y 580.845,Z 631.81,A -85,B 0,C 180,E1 -1904.541,E2 -1904.541} C_VEL
LIN {X 0,Y 580.972,Z 618.525,A -85,B 0,C 180,E1 -1905.344,E2 -1905.344} C_VEL
LIN {X 0,Y 581.201,Z 603.842,A -85,B 0,C 180,E1 -1906.058,E2 -1906.058} C_VEL
LIN {X 0,Y 581.344,Z 589.626,A -85,B 0,C 180,E1 -1906.595,E2 -1906.595} C_VEL
LIN {X 0,Y 581.449,Z 575.2,A -85,B 0,C 180,E1 -1907.001,E2 -1907.001} C_VEL
LIN {X 0,Y 581.517,Z 560.875,A -85,B 0,C 180,E1 -1907.274,E2 -1907.274} C_VEL
LIN {X 0,Y 581.833,Z 403.164,A -85,B 0,C 180,E1 -1909.281,E2 -1909.281} C_VEL
LIN {X 0,Y 580.938,Z 398.282,A -85,B 0,C 180,E1 -1909.392,E2 -1909.392} C_VEL
LIN {X 0,Y 581.229,Z 372.931,A -85,B 0,C 180,E1 -1912.201,E2 -1912.201} C_VEL
LIN {X 0,Y 581.559,Z 347.94,A -85,B 0,C 180,E1 -1915.022,E2 -1915.022} C_VEL
LIN {X 0,Y 581.672,Z 334.153,A -85,B 0,C 180,E1 -1916.607,E2 -1916.607} C_VEL
LIN {X 0,Y 580.325,Z 327.823,A -85,B 0,C 180,E1 -1917.418,E2 -1917.418} C_VEL
LIN {X 0,Y 580.296,Z 327.822,A -85,B 0,C 180,E1 -1920.574,E2 -1920.574} C_VEL
LIN {X 0,Y 580.302,Z 327.829,A -85,B 0,C 180,E1 -1923.316,E2 -1923.316} C_VEL
LIN {X 0,Y 580.247,Z 327.83,A -85,B 0,C 180,E1 -1925.757,E2 -1925.757} C_VEL
LIN {X 0,Y 580.286,Z 327.822,A -85,B 0,C 180,E1 -1928.146,E2 -1928.146} C_VEL
LIN {X 0,Y 580.297,Z 327.823,A -85,B 0,C 180,E1 -1930.843,E2 -1930.843} C_VEL
LIN {X 0,Y 580.285,Z 327.825,A -85,B 0,C 180,E1 -1933.657,E2 -1933.657} C_VEL
LIN {X 0,Y 580.274,Z 327.824,A -85,B 0,C 180,E1 -1936.609,E2 -1936.609} C_VEL
LIN {X 0,Y 580.3,Z 327.829,A -85,B 0,C 180,E1 -1939.157,E2 -1939.157} C_VEL
LIN {X 0,Y 580.288,Z 327.821,A -85,B 0,C 180,E1 -1941.927,E2 -1941.927} C_VEL
LIN {X 0,Y 580.304,Z 327.82,A -85,B 0,C 180,E1 -1944.457,E2 -1944.457} C_VEL
LIN {X 0,Y 580.287,Z 327.828,A -85,B 0,C 180,E1 -1946.975,E2 -1946.975} C_VEL
LIN {X 0,Y 580.294,Z 327.825,A -85,B 0,C 180,E1 -1949.425,E2 -1949.425} C_VEL
LIN {X 0,Y 580.295,Z 327.82,A -85,B 0,C 180,E1 -1952.141,E2 -1952.141} C_VEL
LIN {X 0,Y 580.319,Z 327.824,A -85,B 0,C 180,E1 -1955.27,E2 -1955.27} C_VEL
LIN {X 0,Y 580.27,Z 327.823,A -85,B 0,C 180,E1 -1957.947,E2 -1957.947} C_VEL
LIN {X 0,Y 580.298,Z 327.828,A -85,B 0,C 180,E1 -1960.914,E2 -1960.914} C_VEL
LIN {X 0,Y 580.276,Z 327.823,A -85,B 0,C 180,E1 -1963.826,E2 -1963.826} C_VEL
LIN {X 0,Y 580.324,Z 327.816,A -85,B 0,C 180,E1 -1965.983,E2 -1965.983} C_VEL
LIN {X 0,Y 580.302,Z 327.827,A -85,B 0,C 180,E1 -1968.827,E2 -1968.827} C_VEL
LIN {X 0,Y 580.326,Z 327.817,A -85,B 0,C 180,E1 -1971.644,E2 -1971.644} C_VEL
LIN {X 0,Y 580.329,Z 327.818,A -85,B 0,C 180,E1 -1974.441,E2 -1974.441} C_VEL
LIN {X 0,Y 580.334,Z 327.82,A -85,B 0,C 180,E1 -1977.224,E2 -1977.224} C_VEL
LIN {X 0,Y 580.352,Z 327.813,A -85,B 0,C 180,E1 -1980,E2 -1980} C_VEL
LIN {X 0,Y 580.336,Z 327.823,A -85,B 0,C 180,E1 -1982.777,E2 -1982.777} C_VEL
LIN {X 0,Y 580.324,Z 327.817,A -85,B 0,C 180,E1 -1985.56,E2 -1985.56} C_VEL
LIN {X 0,Y 580.332,Z 327.818,A -85,B 0,C 180,E1 -1988.356,E2 -1988.356} C_VEL
LIN {X 0,Y 580.298,Z 327.824,A -85,B 0,C 180,E1 -1991.191,E2 -1991.191} C_VEL
LIN {X 0,Y 580.324,Z 327.817,A -85,B 0,C 180,E1 -1994.017,E2 -1994.017} C_VEL
LIN {X 0,Y 580.311,Z 327.826,A -85,B 0,C 180,E1 -1996.914,E2 -1996.914} C_VEL
LIN {X 0,Y 580.286,Z 327.821,A -85,B 0,C 180,E1 -1999.823,E2 -1999.823} C_VEL
LIN {X 0,Y 580.281,Z 327.823,A -85,B 0,C 180,E1 -2001.332,E2 -2001.332} C_VEL
LIN {X 0,Y 579.583,Z 327.91,A -85,B 0,C 180,E1 -2001.912,E2 -2001.912} C_VEL
LIN {X 0,Y 576.705,Z 328.276,A -85,B 0,C 180,E1 -2002.851,E2 -2002.851} C_VEL
LIN {X 0,Y 574.311,Z 328.569,A -85,B 0,C 180,E1 -2003.608,E2 -2003.608} C_VEL
LIN {X 0,Y 573.313,Z 328.692,A -85,B 0,C 180,E1 -2004.192,E2 -2004.192} C_VEL
LIN {X 0,Y 573.247,Z 328.703,A -85,B 0,C 180,E1 -2004.389,E2 -2004.389} C_VEL
LIN {X 0,Y 573.207,Z 328.709,A -85,B 0,C 180,E1 -2006.979,E2 -2006.979} C_VEL
LIN {X 0,Y 573.246,Z 328.698,A -85,B 0,C 180,E1 -2009.489,E2 -2009.489} C_VEL
LIN {X 0,Y 573.252,Z 328.707,A -85,B 0,C 180,E1 -2012.646,E2 -2012.646} C_VEL
LIN {X 0,Y 573.252,Z 328.7,A -85,B 0,C 180,E1 -2015.185,E2 -2015.185} C_VEL
LIN {X 0,Y 573.235,Z 328.7,A -85,B 0,C 180,E1 -2017.808,E2 -2017.808} C_VEL
LIN {X 0,Y 573.245,Z 328.707,A -85,B 0,C 180,E1 -2020.526,E2 -2020.526} C_VEL
LIN {X 0,Y 573.208,Z 328.703,A -85,B 0,C 180,E1 -2023.363,E2 -2023.363} C_VEL
LIN {X 0,Y 573.236,Z 328.705,A -85,B 0,C 180,E1 -2026.333,E2 -2026.333} C_VEL
LIN {X 0,Y 573.227,Z 328.711,A -85,B 0,C 180,E1 -2028.543,E2 -2028.543} C_VEL
LIN {X 0,Y 573.237,Z 328.7,A -85,B 0,C 180,E1 -2031.298,E2 -2031.298} C_VEL
LIN {X 0,Y 573.194,Z 328.707,A -85,B 0,C 180,E1 -2034.022,E2 -2034.022} C_VEL
LIN {X 0,Y 573.272,Z 328.705,A -85,B 0,C 180,E1 -2036.518,E2 -2036.518} C_VEL
LIN {X 0,Y 573.222,Z 328.702,A -85,B 0,C 180,E1 -2039.12,E2 -2039.12} C_VEL
LIN {X 0,Y 573.223,Z 328.701,A -85,B 0,C 180,E1 -2041.435,E2 -2041.435} C_VEL
LIN {X 0,Y 573.236,Z 328.707,A -85,B 0,C 180,E1 -2044.589,E2 -2044.589} C_VEL
LIN {X 0,Y 573.222,Z 328.702,A -85,B 0,C 180,E1 -2047.662,E2 -2047.662} C_VEL
LIN {X 0,Y 573.269,Z 328.701,A -85,B 0,C 180,E1 -2050.67,E2 -2050.67} C_VEL
LIN {X 0,Y 573.21,Z 328.703,A -85,B 0,C 180,E1 -2053.621,E2 -2053.621} C_VEL
LIN {X 0,Y 573.26,Z 328.698,A -85,B 0,C 180,E1 -2055.807,E2 -2055.807} C_VEL
LIN {X 0,Y 573.268,Z 328.699,A -85,B 0,C 180,E1 -2058.746,E2 -2058.746} C_VEL
LIN {X 0,Y 573.249,Z 328.698,A -85,B 0,C 180,E1 -2061.54,E2 -2061.54} C_VEL
LIN {X 0,Y 573.274,Z 328.704,A -85,B 0,C 180,E1 -2064.372,E2 -2064.372} C_VEL
LIN {X 0,Y 573.31,Z 328.694,A -85,B 0,C 180,E1 -2067.893,E2 -2067.893} C_VEL
LIN {X 0,Y 573.316,Z 328.693,A -85,B 0,C 180,E1 -2070.703,E2 -2070.703} C_VEL
LIN {X 0,Y 573.279,Z 328.696,A -85,B 0,C 180,E1 -2072.811,E2 -2072.811} C_VEL
LIN {X 0,Y 573.266,Z 328.697,A -85,B 0,C 180,E1 -2075.629,E2 -2075.629} C_VEL
LIN {X 0,Y 573.245,Z 328.704,A -85,B 0,C 180,E1 -2078.46,E2 -2078.46} C_VEL
LIN {X 0,Y 573.24,Z 328.699,A -85,B 0,C 180,E1 -2081.313,E2 -2081.313} C_VEL
LIN {X 0,Y 573.253,Z 328.705,A -85,B 0,C 180,E1 -2084.411,E2 -2084.411} C_VEL
LIN {X 0,Y 573.182,Z 328.709,A -85,B 0,C 180,E1 -2087.114,E2 -2087.114} C_VEL
LIN {X 0,Y 573.255,Z 328.907,A -85,B 0,C 180,E1 -2088.681,E2 -2088.681} C_VEL
LIN {X 0,Y 573.807,Z 333.662,A -85,B 0,C 180,E1 -2089.42,E2 -2089.42} C_VEL
LIN {X 0,Y 573.683,Z 340.452,A -85,B 0,C 180,E1 -2090.435,E2 -2090.435} C_VEL
LIN {X 0,Y 575.17,Z 347.669,A -85,B 0,C 180,E1 -2090.59,E2 -2090.59} C_VEL
LIN {X 0,Y 574.702,Z 505.589,A -85,B 0,C 180,E1 -2092.633,E2 -2092.633} C_VEL
LIN {X 0,Y 574.606,Z 521.397,A -85,B 0,C 180,E1 -2092.994,E2 -2092.994} C_VEL
LIN {X 0,Y 574.427,Z 536.487,A -85,B 0,C 180,E1 -2093.489,E2 -2093.489} C_VEL
LIN {X 0,Y 574.247,Z 550.759,A -85,B 0,C 180,E1 -2094.109,E2 -2094.109} C_VEL
LIN {X 0,Y 574.009,Z 564.24,A -85,B 0,C 180,E1 -2094.842,E2 -2094.842} C_VEL
LIN {X 0,Y 573.817,Z 578.167,A -85,B 0,C 180,E1 -2095.773,E2 -2095.773} C_VEL
LIN {X 0,Y 573.621,Z 589.953,A -85,B 0,C 180,E1 -2096.726,E2 -2096.726} C_VEL
LIN {X 0,Y 573.444,Z 600.698,A -85,B 0,C 180,E1 -2097.757,E2 -2097.757} C_VEL
LIN {X 0,Y 573.297,Z 611.28,A -85,B 0,C 180,E1 -2098.962,E2 -2098.962} C_VEL
LIN {X 0,Y 573.193,Z 620.214,A -85,B 0,C 180,E1 -2100.18,E2 -2100.18} C_VEL
LIN {X 0,Y 573.103,Z 627.781,A -85,B 0,C 180,E1 -2101.412,E2 -2101.412} C_VEL
LIN {X 0,Y 573.034,Z 634.153,A -85,B 0,C 180,E1 -2102.659,E2 -2102.659} C_VEL
LIN {X 0,Y 573.02,Z 639.437,A -85,B 0,C 180,E1 -2103.921,E2 -2103.921} C_VEL
LIN {X 0,Y 572.964,Z 643.642,A -85,B 0,C 180,E1 -2105.205,E2 -2105.205} C_VEL
LIN {X 0,Y 572.938,Z 645.911,A -85,B 0,C 180,E1 -2106.072,E2 -2106.072} C_VEL
LIN {X 0,Y 572.929,Z 648.01,A -85,B 0,C 180,E1 -2107.122,E2 -2107.122} C_VEL
LIN {X 0,Y 572.93,Z 649.566,A -85,B 0,C 180,E1 -2108.272,E2 -2108.272} C_VEL
LIN {X 0,Y 572.924,Z 650.415,A -85,B 0,C 180,E1 -2109.634,E2 -2109.634} C_VEL
LIN {X 0,Y 572.94,Z 650.394,A -85,B 0,C 180,E1 -2110.551,E2 -2110.551} C_VEL
LIN {X 0,Y 572.967,Z 649.835,A -85,B 0,C 180,E1 -2111.563,E2 -2111.563} C_VEL
LIN {X 0,Y 572.962,Z 648.574,A -85,B 0,C 180,E1 -2112.611,E2 -2112.611} C_VEL
LIN {X 0,Y 572.933,Z 646.736,A -85,B 0,C 180,E1 -2113.636,E2 -2113.636} C_VEL
LIN {X 0,Y 572.997,Z 643.37,A -85,B 0,C 180,E1 -2114.975,E2 -2114.975} C_VEL
LIN {X 0,Y 573.01,Z 638.712,A -85,B 0,C 180,E1 -2116.356,E2 -2116.356} C_VEL
LIN {X 0,Y 573.058,Z 632.382,A -85,B 0,C 180,E1 -2117.806,E2 -2117.806} C_VEL
LIN {X 0,Y 573.104,Z 625.965,A -85,B 0,C 180,E1 -2118.998,E2 -2118.998} C_VEL
LIN {X 0,Y 573.245,Z 616.881,A -85,B 0,C 180,E1 -2120.392,E2 -2120.392} C_VEL
LIN {X 0,Y 573.403,Z 606.781,A -85,B 0,C 180,E1 -2121.668,E2 -2121.668} C_VEL
LIN {X 0,Y 573.511,Z 596.064,A -85,B 0,C 180,E1 -2122.801,E2 -2122.801} C_VEL
LIN {X 0,Y 573.74,Z 583.697,A -85,B 0,C 180,E1 -2123.889,E2 -2123.889} C_VEL
LIN {X 0,Y 573.891,Z 572.016,A -85,B 0,C 180,E1 -2124.753,E2 -2124.753} C_VEL
LIN {X 0,Y 574.065,Z 559.333,A -85,B 0,C 180,E1 -2125.533,E2 -2125.533} C_VEL
LIN {X 0,Y 574.324,Z 544.75,A -85,B 0,C 180,E1 -2126.259,E2 -2126.259} C_VEL
LIN {X 0,Y 574.495,Z 530.66,A -85,B 0,C 180,E1 -2126.808,E2 -2126.808} C_VEL
LIN {X 0,Y 574.612,Z 515.573,A -85,B 0,C 180,E1 -2127.246,E2 -2127.246} C_VEL
LIN {X 0,Y 574.74,Z 500.437,A -85,B 0,C 180,E1 -2127.538,E2 -2127.538} C_VEL
LIN {X 0,Y 575.16,Z 347.4,A -85,B 0,C 180,E1 -2129.504,E2 -2129.504} C_VEL
LIN {X 0,Y 573.688,Z 340.424,A -85,B 0,C 180,E1 -2129.659,E2 -2129.659} C_VEL
LIN {X 0,Y 573.777,Z 332.384,A -85,B 0,C 180,E1 -2130.864,E2 -2130.864} C_VEL
LIN {X 0,Y 573.215,Z 328.711,A -85,B 0,C 180,E1 -2131.477,E2 -2131.477} C_VEL
LIN {X 0,Y 573.203,Z 328.707,A -85,B 0,C 180,E1 -2134.587,E2 -2134.587} C_VEL
LIN {X 0,Y 573.197,Z 328.706,A -85,B 0,C 180,E1 -2136.899,E2 -2136.899} C_VEL
LIN {X 0,Y 573.223,Z 328.703,A -85,B 0,C 180,E1 -2139.172,E2 -2139.172} C_VEL
LIN {X 0,Y 573.198,Z 328.708,A -85,B 0,C 180,E1 -2141.41,E2 -2141.41} C_VEL
LIN {X 0,Y 573.209,Z 328.705,A -85,B 0,C 180,E1 -2144.351,E2 -2144.351} C_VEL
LIN {X 0,Y 573.214,Z 328.703,A -85,B 0,C 180,E1 -2146.529,E2 -2146.529} C_VEL
LIN {X 0,Y 573.261,Z 328.702,A -85,B 0,C 180,E1 -2149.403,E2 -2149.403} C_VEL
LIN {X 0,Y 573.223,Z 328.703,A -85,B 0,C 180,E1 -2152.249,E2 -2152.249} C_VEL
LIN {X 0,Y 573.29,Z 328.695,A -85,B 0,C 180,E1 -2155.077,E2 -2155.077} C_VEL
LIN {X 0,Y 573.312,Z 328.695,A -85,B 0,C 180,E1 -2157.892,E2 -2157.892} C_VEL
LIN {X 0,Y 573.316,Z 328.69,A -85,B 0,C 180,E1 -2160.702,E2 -2160.702} C_VEL
LIN {X 0,Y 573.29,Z 328.694,A -85,B 0,C 180,E1 -2162.81,E2 -2162.81} C_VEL
LIN {X 0,Y 573.285,Z 328.701,A -85,B 0,C 180,E1 -2165.628,E2 -2165.628} C_VEL
LIN {X 0,Y 573.254,Z 328.698,A -85,B 0,C 180,E1 -2168.46,E2 -2168.46} C_VEL
LIN {X 0,Y 573.275,Z 328.703,A -85,B 0,C 180,E1 -2171.312,E2 -2171.312} C_VEL
LIN {X 0,Y 573.271,Z 328.695,A -85,B 0,C 180,E1 -2174.419,E2 -2174.419} C_VEL
LIN {X 0,Y 573.261,Z 328.703,A -85,B 0,C 180,E1 -2177.111,E2 -2177.111} C_VEL
LIN {X 0,Y 573.241,Z 328.699,A -85,B 0,C 180,E1 -2180.077,E2 -2180.077} C_VEL
LIN {X 0,Y 573.234,Z 328.7,A -85,B 0,C 180,E1 -2182.338,E2 -2182.338} C_VEL
LIN {X 0,Y 573.251,Z 328.704,A -85,B 0,C 180,E1 -2185.41,E2 -2185.41} C_VEL
LIN {X 0,Y 573.251,Z 328.698,A -85,B 0,C 180,E1 -2188.028,E2 -2188.028} C_VEL
LIN {X 0,Y 573.248,Z 328.698,A -85,B 0,C 180,E1 -2190.176,E2 -2190.176} C_VEL
LIN {X 0,Y 573.254,Z 328.701,A -85,B 0,C 180,E1 -2192.645,E2 -2192.645} C_VEL
LIN {X 0,Y 573.208,Z 328.712,A -85,B 0,C 180,E1 -2195.188,E2 -2195.188} C_VEL
LIN {X 0,Y 573.238,Z 328.7,A -85,B 0,C 180,E1 -2197.807,E2 -2197.807} C_VEL
LIN {X 0,Y 573.246,Z 328.702,A -85,B 0,C 180,E1 -2200.525,E2 -2200.525} C_VEL
LIN {X 0,Y 573.241,Z 328.703,A -85,B 0,C 180,E1 -2203.359,E2 -2203.359} C_VEL
LIN {X 0,Y 573.254,Z 328.7,A -85,B 0,C 180,E1 -2206.33,E2 -2206.33} C_VEL
LIN {X 0,Y 573.261,Z 328.699,A -85,B 0,C 180,E1 -2209.476,E2 -2209.476} C_VEL
LIN {X 0,Y 573.236,Z 328.702,A -85,B 0,C 180,E1 -2212.192,E2 -2212.192} C_VEL
LIN {X 0,Y 573.235,Z 328.704,A -85,B 0,C 180,E1 -2215.229,E2 -2215.229} C_VEL
LIN {X 0,Y 573.25,Z 328.699,A -85,B 0,C 180,E1 -2217.772,E2 -2217.772} C_VEL
LIN {X 0,Y 573.261,Z 328.707,A -85,B 0,C 180,E1 -2220.634,E2 -2220.634} C_VEL
LIN {X 0,Y 573.281,Z 328.873,A -85,B 0,C 180,E1 -2222.408,E2 -2222.408} C_VEL
LIN {X 0,Y 574.91,Z 336.434,A -85,B 0,C 180,E1 -2223.347,E2 -2223.347} C_VEL
LIN {X 0,Y 574.63,Z 359.597,A -85,B 0,C 180,E1 -2226.004,E2 -2226.004} C_VEL
LIN {X 0,Y 574.22,Z 386.314,A -85,B 0,C 180,E1 -2229.029,E2 -2229.029} C_VEL
LIN {X 0,Y 574.042,Z 398.384,A -85,B 0,C 180,E1 -2230.377,E2 -2230.377} C_VEL
LIN {X 0,Y 575.217,Z 405.716,A -85,B 0,C 180,E1 -2230.522,E2 -2230.522} C_VEL
LIN {X 0,Y 574.761,Z 565.056,A -85,B 0,C 180,E1 -2232.581,E2 -2232.581} C_VEL
LIN {X 0,Y 574.607,Z 580.695,A -85,B 0,C 180,E1 -2232.929,E2 -2232.929} C_VEL
LIN {X 0,Y 574.429,Z 596.034,A -85,B 0,C 180,E1 -2233.428,E2 -2233.428} C_VEL
LIN {X 0,Y 574.293,Z 609.763,A -85,B 0,C 180,E1 -2234.017,E2 -2234.017} C_VEL
LIN {X 0,Y 574.049,Z 623.238,A -85,B 0,C 180,E1 -2234.738,E2 -2234.738} C_VEL
LIN {X 0,Y 573.861,Z 636.813,A -85,B 0,C 180,E1 -2235.631,E2 -2235.631} C_VEL
LIN {X 0,Y 573.635,Z 649.346,A -85,B 0,C 180,E1 -2236.629,E2 -2236.629} C_VEL
LIN {X 0,Y 573.478,Z 659.746,A -85,B 0,C 180,E1 -2237.616,E2 -2237.616} C_VEL
LIN {X 0,Y 573.286,Z 669.767,A -85,B 0,C 180,E1 -2238.734,E2 -2238.734} C_VEL
LIN {X 0,Y 573.243,Z 678.855,A -85,B 0,C 180,E1 -2239.938,E2 -2239.938} C_VEL
LIN {X 0,Y 573.132,Z 686.731,A -85,B 0,C 180,E1 -2241.183,E2 -2241.183} C_VEL
LIN {X 0,Y 573.075,Z 694.088,A -85,B 0,C 180,E1 -2242.601,E2 -2242.601} C_VEL
LIN {X 0,Y 573.041,Z 699.922,A -85,B 0,C 180,E1 -2244.016,E2 -2244.016} C_VEL
LIN {X 0,Y 572.951,Z 703.384,A -85,B 0,C 180,E1 -2245.074,E2 -2245.074} C_VEL
LIN {X 0,Y 573.005,Z 706.888,A -85,B 0,C 180,E1 -2246.484,E2 -2246.484} C_VEL
LIN {X 0,Y 572.938,Z 709.192,A -85,B 0,C 180,E1 -2247.891,E2 -2247.891} C_VEL
LIN {X 0,Y 572.936,Z 710.349,A -85,B 0,C 180,E1 -2249.297,E2 -2249.297} C_VEL
LIN {X 0,Y 572.936,Z 710.349,A -85,B 0,C 180,E1 -2250.703,E2 -2250.703} C_VEL
LIN {X 0,Y 572.938,Z 709.191,A -85,B 0,C 180,E1 -2252.109,E2 -2252.109} C_VEL
LIN {X 0,Y 573.005,Z 706.887,A -85,B 0,C 180,E1 -2253.516,E2 -2253.516} C_VEL
LIN {X 0,Y 572.951,Z 703.386,A -85,B 0,C 180,E1 -2254.925,E2 -2254.925} C_VEL
LIN {X 0,Y 573.013,Z 698.61,A -85,B 0,C 180,E1 -2256.337,E2 -2256.337} C_VEL
LIN {X 0,Y 573.093,Z 692.425,A -85,B 0,C 180,E1 -2257.752,E2 -2257.752} C_VEL
LIN {X 0,Y 573.135,Z 684.651,A -85,B 0,C 180,E1 -2259.172,E2 -2259.172} C_VEL
LIN {X 0,Y 573.27,Z 676.371,A -85,B 0,C 180,E1 -2260.418,E2 -2260.418} C_VEL
LIN {X 0,Y 573.385,Z 666.394,A -85,B 0,C 180,E1 -2261.668,E2 -2261.668} C_VEL
LIN {X 0,Y 573.567,Z 656.192,A -85,B 0,C 180,E1 -2262.741,E2 -2262.741} C_VEL
LIN {X 0,Y 573.742,Z 644.023,A -85,B 0,C 180,E1 -2263.819,E2 -2263.819} C_VEL
LIN {X 0,Y 573.959,Z 630.908,A -85,B 0,C 180,E1 -2264.781,E2 -2264.781} C_VEL
LIN {X 0,Y 574.11,Z 618.522,A -85,B 0,C 180,E1 -2265.532,E2 -2265.532} C_VEL
